FUNCTION_BLOCK "Gr050_Code"	// FB 150
TITLE = Gr050 Machine FB44, FB47, FB50, FB51, FB52, FB56, FB88
//COPYRIGHT:    (C) 1999  BUHLER AG, CH-9240 UZWIL, SWITZERLAND
//
//PRODUCT:      DEFAULT
//
//TITLE:        Machine FB44, FB47, FB50, FB51, FB52, FB56, FB88
//                Machine group control
//                Maschinengruppensteuerung
// 
//--------------------------------------------------------------------------------
// 
//IDENT:        AUTHOR:             DEPT:                              DATE:
// 
//P01_FB150.1.0 A_Egli              CT3                                24.Jul.2008
//             1st Release
// 
//--------------------------------------------------------------------------------
// 
//PURPOSE: 
// 
//MANUAL : 
// 
//RESTRICTIONS: 
// 
//--------------------------------------------------------------------------------
//
AUTHOR : EA
FAMILY : USW
VERSION : 9.9
VAR
  Gr : FB 10;	//Standard interface to group
  InOutValue1 : DINT ;	//Data for user
  InOutValue2 : DINT ;	//Data for user
  OutWayConflict : BOOL ;	//Data for user
  OutSelectionOk : BOOL ;	//Data for user
  CmdNewValue : BOOL ;	//Data for user
  CmdNewJob : BOOL ;	//Data for user
  OutCodeOK : BOOL ;	//Data for user
  InEndOfJob : BOOL ;	//Data for user
  staWayOk : BOOL ;	//Data for user
  EdgeStartRelease : BOOL ;	//Data for user
  USW8 : BOOL ;	//Data for user
  USW9 : BOOL ;	//Data for user
  USW10 : BOOL ;	//Data for user
  USW11 : BOOL ;	//Data for user
  USW12 : BOOL ;	//Data for user
  USW13 : BOOL ;	//Data for user
  USW14 : BOOL ;	//Data for user
  USW15 : BOOL ;	//Data for user
  MaFB44 : FB 735;	// Scourer
  MaFB47 : FB 736;	// Pellet
  MaFB48_ALL : FB 709;	// M3HL2
  MaFB48_Carter : FB 710;	// M3HL2
  MaFB48_MTC : FB 711;	// M3HL2
  MaFB48_MTRA : FB 712;	// M3HL2
  MaFB50All : FB 713;	// Motor+6DI
  MaFB50BKT : FB 714;	// Motor+6DI
  MaFB50ELEV : FB 715;	// Motor+6DI
  MaFB50SIEVE : FB 716;	// Motor+6DI
  MaFB51 : FB 718;	// Motor+2DI
  MaFB52 : FB 719;	// Motor+VLS
  MaFB56 : FB 720;	// DischargerA
  _FB56LL : FB 84;	// SubType FB14: DigInpCont
  MaFB50EBM : FB 724;	// Motor+6DI
  MaFB88 : FB 740;	// DischargerFlat
  MaFB88_Door : FB 14;	// DigInpCont
END_VAR
VAR_TEMP
  tmpEnable : BOOL ;
  tmpFlag : BOOL ;
  tmpCmdNext : BOOL ;
  tmpLocal : BOOL ;
  tmpAspOk : BOOL ;
  tmpHWStop : BOOL ;
  tmpInstanzDBNo : INT ;
END_VAR
BEGIN
NETWORK
TITLE =
NETWORK
TITLE = Read command from group control
NETWORK
TITLE = Call Methode Control
// 1. Handle Interface PCControl      
// 2. Prepare mode --> ModePassive,ModeActive,ModeIdling      
// 3. Reset global flags of the group
      CALL  #Gr (
           FcCode                   := 1);
NETWORK
TITLE = Restart Idling Time
      L     #Gr.Par.ParIdling;
      L     2;
      >=I;
      JC    IdTm;
      T     #Gr.Par.ParIdling;
IdTm: NOP   0;
      CLR;
      S     #Gr.CmdRestartIdling;
NETWORK
TITLE = Prepare global flags
NETWORK
TITLE = Set Pattern (Target position)
NETWORK
TITLE = Interlocking WayOk
NETWORK
TITLE = Interlocking Autostart
      CLR;
      R     #Gr.OutAutostart;
NETWORK
TITLE = Interlocking Enable
      A     #Gr.InEnableGr;
      =     #Gr.OutEnableEl;
NETWORK
TITLE = Interlocking Next
      A     #Gr.CmdNext;
      A     #Gr.OutAutostart;
      AN    #Gr.OutNewWay;
      =     #tmpCmdNext;
NETWORK
TITLE = Interlocking Local / HWStop
      A     "PLC_SystemDB".HardwareStop.General;
      =     #tmpHWStop;
      A     #Gr.ModePassive;
      =     #tmpLocal;
NETWORK
TITLE = MaFB44 : Scourer
      NOP   0;
//-InLocal---
      A     #tmpLocal;
      =     DIX [AR2,P#63.4];
//-Interlocking---
      A     #Gr.OutEnableEl;
      =     DIX [AR2,P#62.0];
// 
      A     #tmpCmdNext;
      S     DIX [AR2,P#63.2];
// 
      A     #Gr.OutSeqStop;
      =     DIX [AR2,P#63.7];
// 
//=Values and commands of elements===
//-FB44Level---
//      CLR
//      S     #MaFB44._FB44Level.CmdRunTimeOutTime
// 
//-Read inputs of elements---
      A     I 2.3;
      =     DIX [AR2,P#72.6];
      A     #tmpHWStop;
      =     DIX [AR2,P#74.0];
      A     I 1.3;
      =     DIX [AR2,P#106.6];
      A     #tmpHWStop;
      =     DIX [AR2,P#108.0];
      A     I 1.5;
      =     DIX [AR2,P#140.6];
      A     #tmpHWStop;
      =     DIX [AR2,P#142.0];
      A     I 2.2;
      =     DIX [AR2,P#174.5];
      A     I 2.1;
      =     DIX [AR2,P#174.6];
      A     #tmpHWStop;
      =     DIX [AR2,P#176.0];
      A     I 2.4;
      =     DIX [AR2,P#208.6];
      A     #tmpHWStop;
      =     DIX [AR2,P#210.0];
      A     I 0.4;
      =     DIX [AR2,P#242.6];
      A     #tmpHWStop;
      =     DIX [AR2,P#244.0];
      A     #tmpHWStop;
      =     DIX [AR2,P#278.0];
// 
//-Set Parameters---
// 
//-Call object control---
      BLD   14;
// 
//-Write outputs---
      =     L 10.0;
      L     DINO;
      T     LW 8;
      CDB;
      OPN   DI [LW 8];
      TAR2  LD 4;
      +AR2  P#60.0;
      UC    FB 735;
      LAR2  LD 4;
      CDB;
      BLD   15;
      A     DIX [AR2,P#74.6];
      =     Q 2.4;
      A     DIX [AR2,P#108.6];
      =     Q 1.1;
      A     DIX [AR2,P#142.6];
      =     Q 2.5;
      A     DIX [AR2,P#176.6];
      =     Q 4.1;
      A     DIX [AR2,P#244.6];
      =     Q 0.7;
      A     DIX [AR2,P#278.7];
      =     Q 4.4;
NETWORK
TITLE = MaFB47 : Pellet Cooler
      NOP   0;
//-InLocal---
      A     #tmpLocal;
      =     DIX [AR2,P#311.4];
// 
//-Interlocking---
      A(;
      O     DIX [AR2,P#65.2];
      O     DIX [AR2,P#65.6];
      );
      A     #Gr.OutEnableEl;
      AN    #Gr.OutSeqStop;
      =     DIX [AR2,P#310.0];
// 
      A     #tmpCmdNext;
      S     DIX [AR2,P#311.2];
// 
//-Additional commands---
      CLR;
      =     DIX [AR2,P#310.1];
      =     DIX [AR2,P#310.2];
      =     DIX [AR2,P#310.3];
      =     DIX [AR2,P#310.4];
      S     DIX [AR2,P#310.5];
// 
//=Values and commands of elements===
// 
//-Values and parameters---
      L     0;
      T     DIW [AR2,P#332.0];
//-FB47Level---
//      CLR
//      S     #MaFB47._FB47Level.CmdRunTimeOutTime
// 
//-Read inputs of elements---
      A     #tmpHWStop;
      =     DIX [AR2,P#328.0];
      A     DIX [AR2,P#388.6];
      =     DIX [AR2,P#386.6];
      A     #tmpHWStop;
      =     DIX [AR2,P#388.0];
      A     I 13.3;
      =     DIX [AR2,P#420.6];
      A     #tmpHWStop;
      =     DIX [AR2,P#422.0];
// 
//-Set Parameters---
// 
//-Call object control---
      BLD   14;
// 
//-Write outputs---
      =     L 10.0;
      L     DINO;
      T     LW 8;
      CDB;
      OPN   DI [LW 8];
      TAR2  LD 4;
      +AR2  P#308.0;
      UC    FB 736;
      LAR2  LD 4;
      CDB;
      BLD   15;
      A     DIX [AR2,P#328.7];
      =     #tmpFlag;
NETWORK
TITLE = MaFB48_ALL : 3 Motors and 2 HL
      NOP   0;
//-InLocal---
      A     #tmpLocal;
      =     DIX [AR2,P#455.4];
// 
//-Interlocking---
      A(;
      O     DIX [AR2,P#313.2];
      O     DIX [AR2,P#313.5];
      O     DIX [AR2,P#313.6];
      );
      A     #Gr.OutEnableEl;
      =     DIX [AR2,P#454.0];
// 
      A     #tmpCmdNext;
      S     DIX [AR2,P#455.2];
// 
      A     #Gr.OutSeqStop;
      =     DIX [AR2,P#455.7];
// 
//-Additional commands---
      CLR;
      =     DIX [AR2,P#454.1];
      CLR;
      =     DIX [AR2,P#454.2];
// 
//=Values and commands of elements===
//-FB48HLLow---
//      CLR
//      S     #MaFB48_ALL._FB48HLLow.CmdRunTimeOutTime
//-FB48HLInlet---
//      CLR
//      S     #MaFB48_ALL._FB48HLInlet.CmdRunTimeOutTime
// 
//-Read inputs of elements---
      A     DIX [AR2,P#466.6];
      =     DIX [AR2,P#464.6];
      A     #tmpHWStop;
      =     DIX [AR2,P#466.0];
      A     DIX [AR2,P#500.6];
      =     DIX [AR2,P#498.6];
      A     #tmpHWStop;
      =     DIX [AR2,P#500.0];
      A     DIX [AR2,P#534.6];
      =     DIX [AR2,P#532.6];
      A     #tmpHWStop;
      =     DIX [AR2,P#534.0];
      AN    I 6.7;
      =     DIX [AR2,P#566.6];
      A     #tmpHWStop;
      =     DIX [AR2,P#568.0];
      AN    I 7.5;
      =     DIX [AR2,P#600.6];
      A     #tmpHWStop;
      =     DIX [AR2,P#602.0];
      A     #tmpHWStop;
      =     DIX [AR2,P#636.0];
// 
//-Set Parameters---
// 
//-Call object control---
      BLD   14;
// 
//-Write outputs---
      =     L 10.0;
      L     DINO;
      T     LW 8;
      CDB;
      OPN   DI [LW 8];
      TAR2  LD 4;
      +AR2  P#452.0;
      UC    FB 709;
      LAR2  LD 4;
      CDB;
      BLD   15;
      A     DIX [AR2,P#636.7];
      =     Q 0.1;
NETWORK
TITLE = MaFB48_Carter : 3 Motors and 2 HL
      NOP   0;
//-InLocal---
      A     #tmpLocal;
      =     DIX [AR2,P#669.4];
// 
//-Interlocking---
      A     DIX [AR2,P#457.2];
      A     #Gr.OutEnableEl;
      =     DIX [AR2,P#668.0];
// 
      A     #tmpCmdNext;
      S     DIX [AR2,P#669.2];
// 
      A     #Gr.OutSeqStop;
      =     DIX [AR2,P#669.7];
// 
//-Additional commands---
      CLR;
      =     DIX [AR2,P#668.1];
      CLR;
      =     DIX [AR2,P#668.2];
// 
//=Values and commands of elements===
//-FB48HLLow_C---
//      CLR
//      S     #MaFB48_Carter._FB48HLLow_C.CmdRunTimeOutTime
//-FB48HLInlet_C---
//      CLR
//      S     #MaFB48_Carter._FB48HLInlet_C.CmdRunTimeOutTime
// 
//-Read inputs of elements---
      A     I 10.0;
      =     DIX [AR2,P#678.6];
      A     #tmpHWStop;
      =     DIX [AR2,P#680.0];
      A     I 9.7;
      =     DIX [AR2,P#712.6];
      A     #tmpHWStop;
      =     DIX [AR2,P#714.0];
      A     I 12.3;
      =     DIX [AR2,P#746.6];
      A     #tmpHWStop;
      =     DIX [AR2,P#748.0];
      AN    I 6.6;
      =     DIX [AR2,P#780.6];
      A     #tmpHWStop;
      =     DIX [AR2,P#782.0];
      AN    I 8.0;
      =     DIX [AR2,P#814.6];
      A     #tmpHWStop;
      =     DIX [AR2,P#816.0];
      A     #tmpHWStop;
      =     DIX [AR2,P#850.0];
// 
//-Set Parameters---
// 
//-Call object control---
      BLD   14;
// 
//-Write outputs---
      =     L 10.0;
      L     DINO;
      T     LW 8;
      CDB;
      OPN   DI [LW 8];
      TAR2  LD 4;
      +AR2  P#666.0;
      UC    FB 710;
      LAR2  LD 4;
      CDB;
      BLD   15;
      A     DIX [AR2,P#680.6];
      =     Q 4.3;
      A     DIX [AR2,P#714.6];
      =     Q 4.6;
      A     DIX [AR2,P#748.6];
      =     Q 5.1;
      A     DIX [AR2,P#850.7];
      =     Q 0.1;
NETWORK
TITLE = MaFB48_MTC : 3 Motors and 2 HL
      NOP   0;
//-InLocal---
      A     #tmpLocal;
      =     DIX [AR2,P#883.4];
// 
//-Interlocking---
      A     DIX [AR2,P#671.2];
      A     #Gr.OutEnableEl;
      =     DIX [AR2,P#882.0];
// 
      A     #tmpCmdNext;
      S     DIX [AR2,P#883.2];
// 
      A     #Gr.OutSeqStop;
      =     DIX [AR2,P#883.7];
// 
//-Additional commands---
      CLR;
      =     DIX [AR2,P#882.1];
      CLR;
      =     DIX [AR2,P#882.2];
// 
//=Values and commands of elements===
//-FB48HLLow---
//      CLR
//      S     #MaFB48_MTC._FB48HLLow.CmdRunTimeOutTime
//-FB48HLInletMTC---
//      CLR
//      S     #MaFB48_MTC._FB48HLInletMTC.CmdRunTimeOutTime
// 
//-Read inputs of elements---
      A     I 7.7;
      =     DIX [AR2,P#892.6];
      A     #tmpHWStop;
      =     DIX [AR2,P#894.0];
      A     I 12.7;
      =     DIX [AR2,P#926.6];
      A     #tmpHWStop;
      =     DIX [AR2,P#928.0];
      A     I 8.1;
      =     DIX [AR2,P#960.6];
      A     #tmpHWStop;
      =     DIX [AR2,P#962.0];
      AN    I 6.7;
      =     DIX [AR2,P#994.6];
      A     #tmpHWStop;
      =     DIX [AR2,P#996.0];
      AN    I 7.6;
      =     DIX [AR2,P#1028.6];
      A     #tmpHWStop;
      =     DIX [AR2,P#1030.0];
      A     #tmpHWStop;
      =     DIX [AR2,P#1064.0];
// 
//-Set Parameters---
// 
//-Call object control---
      BLD   14;
// 
//-Write outputs---
      =     L 10.0;
      L     DINO;
      T     LW 8;
      CDB;
      OPN   DI [LW 8];
      TAR2  LD 4;
      +AR2  P#880.0;
      UC    FB 711;
      LAR2  LD 4;
      CDB;
      BLD   15;
      A     DIX [AR2,P#894.6];
      =     Q 4.2;
      A     DIX [AR2,P#928.6];
      =     Q 5.2;
      A     DIX [AR2,P#962.6];
      =     Q 3.0;
      A     DIX [AR2,P#1064.7];
      =     Q 0.1;
NETWORK
TITLE = MaFB48_MTRA : 3 Motors and 2 HL
      NOP   0;
//-InLocal---
      A     #tmpLocal;
      =     DIX [AR2,P#1097.4];
// 
//-Interlocking---
      A     DIX [AR2,P#885.2];
      A     #Gr.OutEnableEl;
      =     DIX [AR2,P#1096.0];
// 
      A     #tmpCmdNext;
      S     DIX [AR2,P#1097.2];
// 
      A     #Gr.OutSeqStop;
      =     DIX [AR2,P#1097.7];
// 
//-Additional commands---
      CLR;
      =     DIX [AR2,P#1096.1];
      CLR;
      =     DIX [AR2,P#1096.2];
// 
//=Values and commands of elements===
//-FB48HLInletMTRA---
//      CLR
//      S     #MaFB48_MTRA._FB48HLInletMTRA.CmdRunTimeOutTime
// 
//-Read inputs of elements---
      A     I 12.5;
      =     DIX [AR2,P#1106.6];
      A     #tmpHWStop;
      =     DIX [AR2,P#1108.0];
      A     I 8.3;
      =     DIX [AR2,P#1140.6];
      A     #tmpHWStop;
      =     DIX [AR2,P#1142.0];
      A     DIX [AR2,P#1176.6];
      =     DIX [AR2,P#1174.6];
      A     #tmpHWStop;
      =     DIX [AR2,P#1176.0];
      AN    I 7.4;
      =     DIX [AR2,P#1242.6];
      A     #tmpHWStop;
      =     DIX [AR2,P#1244.0];
// 
//-Set Parameters---
// 
//-Call object control---
      BLD   14;
// 
//-Write outputs---
      =     L 10.0;
      L     DINO;
      T     LW 8;
      CDB;
      OPN   DI [LW 8];
      TAR2  LD 4;
      +AR2  P#1094.0;
      UC    FB 712;
      LAR2  LD 4;
      CDB;
      BLD   15;
      A     DIX [AR2,P#1108.6];
      =     Q 5.0;
      A     DIX [AR2,P#1142.6];
      =     Q 3.1;
NETWORK
TITLE = MaFB50All : Motor + 4 digiatl inputs     
      NOP   0;
//-InLocal---
      A     #tmpLocal;
      =     DIX [AR2,P#1311.4];
//-Interlocking---
      A     DIX [AR2,P#1099.2];
      A     #Gr.OutEnableEl;
      =     DIX [AR2,P#1310.1];
      A     #tmpCmdNext;
      S     DIX [AR2,P#1311.2];
      A     #Gr.OutSeqStop;
      =     DIX [AR2,P#1311.7];
// 
//=Values and commands of elements===
//-FB50Mon1---
//      CLR
//      S     #MaFB50All._FB50Mon1.CmdRunTimeOutTime
//-FB50Mon2---
//      CLR
//      S     #MaFB50All._FB50Mon2.CmdRunTimeOutTime
//-FB50Mon3---
//      CLR
//      S     #MaFB50All._FB50Mon3.CmdRunTimeOutTime
//-FB50MonInlet---
//      CLR
//      S     #MaFB50All._FB50MonInlet.CmdRunTimeOutTime
// 
//-Read inputs of elements---
      A     I 22.0;
      =     DIX [AR2,P#1322.6];
      A     #tmpHWStop;
      =     DIX [AR2,P#1324.0];
      A     I 22.1;
      =     DIX [AR2,P#1356.6];
      A     #tmpHWStop;
      =     DIX [AR2,P#1358.0];
      A     I 22.2;
      =     DIX [AR2,P#1390.6];
      A     #tmpHWStop;
      =     DIX [AR2,P#1392.0];
      A     I 22.3;
      =     DIX [AR2,P#1424.6];
      A     #tmpHWStop;
      =     DIX [AR2,P#1426.0];
      A     I 22.4;
      =     DIX [AR2,P#1526.6];
      A     I 22.5;
      =     DIX [AR2,P#1526.5];
      A     #tmpHWStop;
      =     DIX [AR2,P#1528.0];
// 
//-Set Parameters---
// 
//-Call object control---
      BLD   14;
// 
//-Write outputs---
      =     L 10.0;
      L     DINO;
      T     LW 8;
      CDB;
      OPN   DI [LW 8];
      TAR2  LD 4;
      +AR2  P#1308.0;
      UC    FB 713;
      LAR2  LD 4;
      CDB;
      BLD   15;
      A     DIX [AR2,P#1528.6];
      =     Q 22.4;
      A     DIX [AR2,P#1528.5];
      =     Q 22.5;
NETWORK
TITLE = MaFB50BKT : Motor + 4 digiatl inputs
      NOP   0;
//-InLocal---
      A     #tmpLocal;
      =     DIX [AR2,P#1561.4];
//-Interlocking---
      A     DIX [AR2,P#1313.2];
      A     #Gr.OutEnableEl;
      =     DIX [AR2,P#1560.1];
      A     #tmpCmdNext;
      S     DIX [AR2,P#1561.2];
      A     #Gr.OutSeqStop;
      =     DIX [AR2,P#1561.7];
// 
//=Values and commands of elements===
//-FB50LSBKT---
//      CLR
//      S     #MaFB50BKT._FB50LSBKT.CmdRunTimeOutTime
//-FB50SM1BKT---
//      CLR
//      S     #MaFB50BKT._FB50SM1BKT.CmdRunTimeOutTime
//-FB50SM2BKT---
//      CLR
//      S     #MaFB50BKT._FB50SM2BKT.CmdRunTimeOutTime
//-FB50HLBKT---
//      CLR
//      S     #MaFB50BKT._FB50HLBKT.CmdRunTimeOutTime
// 
//-Read inputs of elements---
      A     I 13.5;
      =     DIX [AR2,P#1572.6];
      A     #tmpHWStop;
      =     DIX [AR2,P#1574.0];
      A     I 1.4;
      =     DIX [AR2,P#1606.6];
      A     #tmpHWStop;
      =     DIX [AR2,P#1608.0];
      A     I 1.2;
      =     DIX [AR2,P#1640.6];
      A     #tmpHWStop;
      =     DIX [AR2,P#1642.0];
      A     I 8.2;
      =     DIX [AR2,P#1674.6];
      A     #tmpHWStop;
      =     DIX [AR2,P#1676.0];
      A     I 12.4;
      =     DIX [AR2,P#1776.6];
      A     I 12.2;
      =     DIX [AR2,P#1776.5];
      A     #tmpHWStop;
      =     DIX [AR2,P#1778.0];
// 
//-Set Parameters---
// 
//-Call object control---
      BLD   14;
// 
//-Write outputs---
      =     L 10.0;
      L     DINO;
      T     LW 8;
      CDB;
      OPN   DI [LW 8];
      TAR2  LD 4;
      +AR2  P#1558.0;
      UC    FB 714;
      LAR2  LD 4;
      CDB;
      BLD   15;
      A     DIX [AR2,P#1778.6];
      =     Q 3.4;
      A     DIX [AR2,P#1778.5];
      =     Q 3.5;
NETWORK
TITLE = MaFB50SIEVE : Motor + 4 digiatl inputs
      NOP   0;
//-InLocal---
      A     #tmpLocal;
      =     DIX [AR2,P#2061.4];
//-Interlocking---
      A     DIX [AR2,P#1563.2];
      A     #Gr.OutEnableEl;
      =     DIX [AR2,P#2060.1];
      A     #tmpCmdNext;
      S     DIX [AR2,P#2061.2];
      A     #Gr.OutSeqStop;
      =     DIX [AR2,P#2061.7];
// 
//=Values and commands of elements===
//-FB50HL_Waste---
//      CLR
//      S     #MaFB50SIEVE._FB50HL_Waste.CmdRunTimeOutTime
//-FB50LSA---
//      CLR
//      S     #MaFB50SIEVE._FB50LSA.CmdRunTimeOutTime
//-FB50LSB---
//      CLR
//      S     #MaFB50SIEVE._FB50LSB.CmdRunTimeOutTime
//-FB50HL_Sieve---
//      CLR
//      S     #MaFB50SIEVE._FB50HL_Sieve.CmdRunTimeOutTime
// 
//-Read inputs of elements---
      A     I 28.5;
      =     DIX [AR2,P#2072.6];
      A     #tmpHWStop;
      =     DIX [AR2,P#2074.0];
      A     I 9.5;
      =     DIX [AR2,P#2106.6];
      A     #tmpHWStop;
      =     DIX [AR2,P#2108.0];
      A     I 0.0;
      =     DIX [AR2,P#2140.6];
      A     #tmpHWStop;
      =     DIX [AR2,P#2142.0];
      A     I 8.6;
      =     DIX [AR2,P#2174.6];
      A     #tmpHWStop;
      =     DIX [AR2,P#2176.0];
      A     I 10.3;
      =     DIX [AR2,P#2276.6];
      A     I 10.1;
      =     DIX [AR2,P#2276.5];
      A     #tmpHWStop;
      =     DIX [AR2,P#2278.0];
// 
//-Set Parameters---
// 
//-Call object control---
      BLD   14;
// 
//-Write outputs---
      =     L 10.0;
      L     DINO;
      T     LW 8;
      CDB;
      OPN   DI [LW 8];
      TAR2  LD 4;
      +AR2  P#2058.0;
      UC    FB 716;
      LAR2  LD 4;
      CDB;
      BLD   15;
      A     DIX [AR2,P#2278.6];
      =     Q 3.6;
      A     DIX [AR2,P#2278.5];
      =     Q 3.3;
NETWORK
TITLE = MaFB51 : Motor with 2 digital input
      NOP   0;
//-InLocal---
      A     #tmpLocal;
      =     DIX [AR2,P#2311.4];
// 
//-Interlocking---
      A     #Gr.OutEnableEl;
      =     DIX [AR2,P#2310.1];
// 
      A     DIX [AR2,P#2063.2];
      A     #tmpCmdNext;
      S     DIX [AR2,P#2311.2];
// 
      A     #Gr.OutSeqStop;
      =     DIX [AR2,P#2311.7];
// 
//=Values and commands of elements===
//-FB51Mon1---
//      CLR
//      S     #MaFB51._FB51Mon1.CmdRunTimeOutTime
//-FB51Mon2---
//      CLR
//      S     #MaFB51._FB51Mon2.CmdRunTimeOutTime
// 
//-Read inputs of elements---
      AN    I 0.3;
      =     DIX [AR2,P#2320.6];
      A     #tmpHWStop;
      =     DIX [AR2,P#2322.0];
      AN    I 0.5;
      =     DIX [AR2,P#2354.6];
      A     #tmpHWStop;
      =     DIX [AR2,P#2356.0];
// 
//-Set Parameters---
// 
//-Call object control---
      BLD   14;
// 
//-Write outputs---
      =     L 10.0;
      L     DINO;
      T     LW 8;
      CDB;
      OPN   DI [LW 8];
      TAR2  LD 4;
      +AR2  P#2308.0;
      UC    FB 718;
      LAR2  LD 4;
      CDB;
      BLD   15;
NETWORK
TITLE = MaFB52 : Motor with Bypass flap
      NOP   0;
//-InLocal---
      A     #tmpLocal;
      =     DIX [AR2,P#2423.4];
//-Interlocking---
      A     #Gr.OutEnableEl;
      =     DIX [AR2,P#2422.1];
      A     #tmpCmdNext;
      S     DIX [AR2,P#2423.2];
      A     #Gr.OutSeqStop;
      =     DIX [AR2,P#2423.7];
      A     "ENG_RemarkFlag";
      =     DIX [AR2,P#2422.4];
//-Additional commands---
      CLR;
      =     DIX [AR2,P#2422.2];
      =     DIX [AR2,P#2422.3];
// 
//=Values and commands of elements===
//-FB52Mon1---
//      CLR
//      S     #MaFB52._FB52Mon1.CmdRunTimeOutTime
//-FB52HLInlet---
//      CLR
//      S     #MaFB52._FB52HLInlet.CmdRunTimeOutTime
// 
//-Read inputs of elements---
      A     I 52.1;
      =     DIX [AR2,P#2438.6];
      A     #tmpHWStop;
      =     DIX [AR2,P#2440.0];
      A     I 33.4;
      =     DIX [AR2,P#2472.6];
      A     I 33.3;
      =     DIX [AR2,P#2472.5];
      A     #tmpHWStop;
      =     DIX [AR2,P#2474.0];
      A     I 52.3;
      =     DIX [AR2,P#2506.5];
      A     I 52.4;
      =     DIX [AR2,P#2506.6];
      A     #tmpHWStop;
      =     DIX [AR2,P#2508.0];
      AN    I 52.0;
      =     DIX [AR2,P#2540.6];
      A     #tmpHWStop;
      =     DIX [AR2,P#2542.0];
      A     I 52.6;
      =     DIX [AR2,P#2574.5];
      A     I 52.7;
      =     DIX [AR2,P#2574.6];
      A     #tmpHWStop;
      =     DIX [AR2,P#2576.0];
      A     #tmpHWStop;
      =     DIX [AR2,P#2610.0];
// 
//-Set Parameters---
// 
//-Call object control---
      BLD   14;
// 
//-Write outputs---
      =     L 10.0;
      L     DINO;
      T     LW 8;
      CDB;
      OPN   DI [LW 8];
      TAR2  LD 4;
      +AR2  P#2420.0;
      UC    FB 719;
      LAR2  LD 4;
      CDB;
      BLD   15;
      A     DIX [AR2,P#2474.6];
      =     Q 36.4;
      A     DIX [AR2,P#2474.5];
      =     Q 36.3;
      A     DIX [AR2,P#2508.5];
      =     Q 52.3;
      A     DIX [AR2,P#2508.6];
      =     Q 52.4;
      A     DIX [AR2,P#2576.5];
      =     Q 52.6;
      A     DIX [AR2,P#2576.6];
      =     Q 52.7;
NETWORK
TITLE = MaFB56 : Bin Discharger A
      NOP   0;
//-InLocal---
      A     #tmpLocal;
      =     DIX [AR2,P#2643.4];
// 
//-Interlocking---
      A     #Gr.OutEnableEl;
      AN    #Gr.OutSeqStop;
      =     DIX [AR2,P#2642.0];
// 
      A     #tmpCmdNext;
      S     DIX [AR2,P#2643.2];
// 
//=Additional commands and signals===
//-Bin emptying---
      CLR;
      =     DIX [AR2,P#2642.1];
//-Low Level---
      A     DIX [AR2,P#2769.0];
      O     DIX [AR2,P#2769.1];
      O     DIX [AR2,P#2769.4];
      =     DIX [AR2,P#2642.3];
      A     DIX [AR2,P#2769.2];
      =     DIX [AR2,P#2642.4];
// 
//=Values and commands of elements===
//-FB56LS---
//      CLR
//      S     #MaFB56._FB56LS.CmdRunTimeOutTime
// 
//-Read inputs of elements---
      A     I 33.6;
      =     DIX [AR2,P#2664.6];
      A     I 34.1;
      =     DIX [AR2,P#2664.5];
      A     I 34.0;
      =     DIX [AR2,P#2664.3];
      A     I 33.7;
      =     DIX [AR2,P#2664.4];
      A     #tmpHWStop;
      =     DIX [AR2,P#2666.0];
      A     I 34.2;
      =     DIX [AR2,P#2698.6];
      A     #tmpHWStop;
      =     DIX [AR2,P#2700.0];
      A     #tmpHWStop;
      =     DIX [AR2,P#2734.0];
// 
//-Set Parameters---
// 
//-Call object control---
      BLD   14;
// 
//-Write outputs---
      =     L 10.0;
      L     DINO;
      T     LW 8;
      CDB;
      OPN   DI [LW 8];
      TAR2  LD 4;
      +AR2  P#2640.0;
      UC    FB 720;
      LAR2  LD 4;
      CDB;
      BLD   15;
      A     DIX [AR2,P#2666.6];
      =     Q 36.1;
      A     DIX [AR2,P#2666.5];
      =     Q 35.0;
      A     DIX [AR2,P#2666.3];
      =     Q 36.0;
      A     DIX [AR2,P#2666.4];
      =     Q 36.2;
      A     DIX [AR2,P#2700.6];
      =     Q 35.3;
NETWORK
TITLE = FB56LL : 
      NOP   0;
//-Local---
      SET;
      =     DIX [AR2,P#2767.4];
// 
//-Monitoring---
// 
//-Read inputs---
      A     #tmpHWStop;
      =     DIX [AR2,P#2768.0];
// 
//-Set Parameters---
// 
//-Call object control---
      BLD   14;
// 
//-Write outputs---
      =     L 10.0;
      L     DINO;
      T     LW 8;
      CDB;
      OPN   DI [LW 8];
      TAR2  LD 4;
      +AR2  P#2764.0;
      UC    "GCS7_E_Level";
      LAR2  LD 4;
      CDB;
      BLD   15;
NETWORK
TITLE = MaFB50ELEV : Motor + 4 digiatl inputs 
      NOP   0;
//-InLocal---
      A     #tmpLocal;
      =     DIX [AR2,P#1811.4];
//-Interlocking---
      A     DIX [AR2,P#2645.2];
      A     #Gr.OutEnableEl;
      =     DIX [AR2,P#1810.1];
      A     #tmpCmdNext;
      S     DIX [AR2,P#1811.2];
      A     #Gr.OutSeqStop;
      =     DIX [AR2,P#1811.7];
// 
//=Values and commands of elements===
//-FB50BM1---
//      CLR
//      S     #MaFB50ELEV._FB50BM1.CmdRunTimeOutTime
//-FB50BM2---
//      CLR
//      S     #MaFB50ELEV._FB50BM2.CmdRunTimeOutTime
//-FB50SM_ELEV---
//      CLR
//      S     #MaFB50ELEV._FB50SM_ELEV.CmdRunTimeOutTime
// 
//-Read inputs of elements---
      A     I 9.0;
      =     DIX [AR2,P#1856.6];
      A     #tmpHWStop;
      =     DIX [AR2,P#1858.0];
      A     I 8.7;
      =     DIX [AR2,P#1890.6];
      A     #tmpHWStop;
      =     DIX [AR2,P#1892.0];
      A     I 2.5;
      =     DIX [AR2,P#1924.6];
      A     #tmpHWStop;
      =     DIX [AR2,P#1926.0];
      A     I 12.6;
      =     DIX [AR2,P#2026.6];
      A     I 13.4;
      =     DIX [AR2,P#2026.5];
      A     #tmpHWStop;
      =     DIX [AR2,P#2028.0];
// 
//-Set Parameters---
// 
//-Call object control---
      BLD   14;
// 
//-Write outputs---
      =     L 10.0;
      L     DINO;
      T     LW 8;
      CDB;
      OPN   DI [LW 8];
      TAR2  LD 4;
      +AR2  P#1808.0;
      UC    FB 715;
      LAR2  LD 4;
      CDB;
      BLD   15;
      A     DIX [AR2,P#2028.6];
      =     Q 13.7;
      A     DIX [AR2,P#2028.5];
      =     Q 14.4;
NETWORK
TITLE = MaFB50EBM : Elevator mit EBM
      NOP   0;
//-Read Inputs of Machine---
      A     I 150.0;
      =     DIX [AR2,P#2800.6];
//-InLocal---
      A     #tmpLocal;
      =     DIX [AR2,P#2801.4];
//-Interlocking---
      A     DIX [AR2,P#1813.2];
      A     #Gr.OutEnableEl;
      =     DIX [AR2,P#2800.1];
      A     #tmpCmdNext;
      S     DIX [AR2,P#2801.2];
      A     #Gr.OutSeqStop;
      =     DIX [AR2,P#2801.7];
// 
//-Additional commands---
      A     DIX [AR2,P#2848.6];
      O     DIX [AR2,P#2882.6];
      O     DIX [AR2,P#2916.6];
      O     DIX [AR2,P#2950.6];
      O     DIX [AR2,P#2984.6];
      A(;
      O     DIX [AR2,P#3017.5];
      O     DIX [AR2,P#2801.4];
      );
      A     DIX [AR2,P#2803.4];
      S     DIX [AR2,P#2801.3];
// 
//=Values and commands of elements===
//-MaFB50BMTop1---
//      CLR
//      S     #MaFB50EBM.MaFB50BMTop1.CmdRunTimeOutTime
//-MaFB50BMTop2---
//      CLR
//      S     #MaFB50EBM.MaFB50BMTop2.CmdRunTimeOutTime
//-MaFB50BMBottom1---
//      CLR
//      S     #MaFB50EBM.MaFB50BMBottom1.CmdRunTimeOutTime
//-MaFB50BMBottom2---
//      CLR
//      S     #MaFB50EBM.MaFB50BMBottom2.CmdRunTimeOutTime
//-MaFB50SM---
//      CLR
//      S     #MaFB50EBM.MaFB50SM.CmdRunTimeOutTime
// 
//-Read inputs of elements---
      A     I 150.1;
      =     DIX [AR2,P#2846.6];
      A     #tmpHWStop;
      =     DIX [AR2,P#2848.0];
      A     I 150.2;
      =     DIX [AR2,P#2880.6];
      A     #tmpHWStop;
      =     DIX [AR2,P#2882.0];
      A     I 150.4;
      =     DIX [AR2,P#2914.6];
      A     #tmpHWStop;
      =     DIX [AR2,P#2916.0];
      A     I 150.5;
      =     DIX [AR2,P#2948.6];
      A     #tmpHWStop;
      =     DIX [AR2,P#2950.0];
      A     I 150.3;
      =     DIX [AR2,P#2982.6];
      A     #tmpHWStop;
      =     DIX [AR2,P#2984.0];
      A     I 149.0;
      =     DIX [AR2,P#3016.6];
      A     #tmpHWStop;
      =     DIX [AR2,P#3018.0];
// 
//-Set Parameters---
// 
//-Call object control---
      BLD   14;
// 
//-Write outputs---
      =     L 10.0;
      L     DINO;
      T     LW 8;
      CDB;
      OPN   DI [LW 8];
      TAR2  LD 4;
      +AR2  P#2798.0;
      UC    FB 724;
// 
      LAR2  LD 4;
      CDB;
      BLD   15;
      A     DIX [AR2,P#2802.7];
      =     Q 150.0;
      A     DIX [AR2,P#2802.4];
      =     Q 150.1;
      A     DIX [AR2,P#2802.5];
// 
      =     Q 150.2;
      A     DIX [AR2,P#2802.6];
      =     Q 150.3;
      AN    DIX [AR2,P#2849.4];
      AN    DIX [AR2,P#2883.4];
      AN    DIX [AR2,P#2917.4];
      AN    DIX [AR2,P#2951.4];
      AN    DIX [AR2,P#2985.4];
      ON    DIX [AR2,P#2801.4];
      O     DIX [AR2,P#3017.5];
      =     Q 150.4;
      A     DIX [AR2,P#3018.6];
      =     Q 149.0;
NETWORK
TITLE = MaFB88_Door : Bin Discharger Flat-Bottom
      NOP   0;
//-InLocal---
      A     #tmpLocal;
      =     DIX [AR2,P#3343.4];
// 
//-Monitoring---
      SET;
      =     DIX [AR2,P#3342.0];
      CLR;
      =     DIX [AR2,P#3342.1];
// 
//-PreAlarm---
      CLR;
      =     DIX [AR2,P#3342.2];
      CLR;
      =     DIX [AR2,P#3342.3];
// 
//-Additional commands---
//      CLR
//      S     #MaFB88_Door.CmdRunTimeOutTime
// 
//-Read inputs---
      A     I 96.2;
      =     DIX [AR2,P#3342.6];
      A     #tmpHWStop;
      =     DIX [AR2,P#3344.0];
// 
//-Set Parameters---
// 
//-Call object control---
      BLD   14;
// 
//-Write outputs---
      =     L 10.0;
      L     DINO;
      T     LW 8;
      CDB;
      OPN   DI [LW 8];
      TAR2  LD 4;
      +AR2  P#3340.0;
      UC    "GCS7_E_DigInput";
      LAR2  LD 4;
      CDB;
      BLD   15;
NETWORK
TITLE = MaFB88 : Bin Discharger Flat-Bottom  
      NOP   0;
//-InLocal---
// 
//-Interlocking---
// 
      SET;
      S     DIX [AR2,P#3051.2];
// 
//=Additional commands and signals===
//-Bin emptying---
//-LSDorr---
      A     DIX [AR2,P#3345.0];
      =     DIX [AR2,P#3050.6];
      A     DIX [AR2,P#3345.2];
      =     DIX [AR2,P#3050.5];
// 
//=Values and commands of elements===
//-MaFB88_LL---
//      CLR
//      S     #MaFB88.MaFB88_LL.CmdRunTimeOutTime
//-MaFB88_Switch---
//      CLR
//      S     #MaFB88.MaFB88_Switch.CmdRunTimeOutTime
// 
//-Read inputs of elements---
      A     I 95.0;
      =     DIX [AR2,P#3070.5];
      A     I 95.1;
      =     DIX [AR2,P#3070.6];
      A     #tmpHWStop;
      =     DIX [AR2,P#3072.0];
      A     #tmpHWStop;
      =     DIX [AR2,P#3106.0];
      A     I 96.5;
      =     DIX [AR2,P#3104.6];
      A     I 96.3;
      =     DIX [AR2,P#3138.6];
      A     #tmpHWStop;
      =     DIX [AR2,P#3140.0];
      A     I 96.4;
      =     DIX [AR2,P#3172.6];
      A     #tmpHWStop;
      =     DIX [AR2,P#3174.0];
      A     I 95.2;
      =     DIX [AR2,P#3206.5];
      A     I 95.3;
      =     DIX [AR2,P#3206.6];
      A     #tmpHWStop;
      =     DIX [AR2,P#3208.0];
      A     I 95.4;
      =     DIX [AR2,P#3240.5];
      A     I 95.5;
      =     DIX [AR2,P#3240.6];
      A     #tmpHWStop;
      =     DIX [AR2,P#3242.0];
      A     I 95.6;
      =     DIX [AR2,P#3274.5];
      A     I 95.7;
      =     DIX [AR2,P#3274.6];
      A     #tmpHWStop;
      =     DIX [AR2,P#3276.0];
      A     I 96.0;
      =     DIX [AR2,P#3308.5];
      A     I 96.1;
      =     DIX [AR2,P#3308.6];
      A     #tmpHWStop;
      =     DIX [AR2,P#3310.0];
// 
//-Set Parameters---
// 
//-Call object control---
      BLD   14;
// 
//-Write outputs---
      =     L 10.0;
      L     DINO;
      T     LW 8;
      CDB;
      OPN   DI [LW 8];
      TAR2  LD 4;
      +AR2  P#3048.0;
      UC    FB 740;
      LAR2  LD 4;
      CDB;
      BLD   15;
      A     DIX [AR2,P#3072.6];
      =     Q 95.0;
      A     DIX [AR2,P#3140.6];
      =     Q 96.3;
NETWORK
TITLE = Test Fault
      A     DIX [AR2,P#65.4];
      O     DIX [AR2,P#313.4];
      O     DIX [AR2,P#457.4];
      O     DIX [AR2,P#671.4];
      O     DIX [AR2,P#885.4];
      O     DIX [AR2,P#1099.4];
      O     DIX [AR2,P#1313.4];
      O     DIX [AR2,P#1563.4];
      O     DIX [AR2,P#2063.4];
      O     DIX [AR2,P#2313.4];
      O     DIX [AR2,P#2425.4];
      O     DIX [AR2,P#2645.4];
      O     DIX [AR2,P#2769.4];
      O     DIX [AR2,P#1813.4];
      O     DIX [AR2,P#2803.4];
      O     DIX [AR2,P#3345.4];
      O     DIX [AR2,P#3053.4];
      =     #Gr.VarFault;
NETWORK
TITLE = Test Warning
      A     DIX [AR2,P#2312.0];
      =     #Gr.OutWarning;
NETWORK
TITLE = Test Stopped
      A     DIX [AR2,P#65.0];
      A(;
      O     DIX [AR2,P#313.0];
      O     DIX [AR2,P#313.6];
      );
      A     DIX [AR2,P#457.0];
      A     DIX [AR2,P#671.0];
      A     DIX [AR2,P#885.0];
      A     DIX [AR2,P#1099.0];
      A     DIX [AR2,P#1313.0];
      A     DIX [AR2,P#1563.0];
      A     DIX [AR2,P#2063.0];
      A     DIX [AR2,P#2313.0];
      A(;
      AN    DIX [AR2,P#2422.1];
      O     DIX [AR2,P#2423.7];
      A     DIX [AR2,P#2425.6];
      O     DIX [AR2,P#2425.0];
      );
      A     DIX [AR2,P#2645.0];
      A     DIX [AR2,P#1813.0];
      A     DIX [AR2,P#2803.0];
      A     DIX [AR2,P#3053.0];
      AN    #Gr.VarFault;
      =     #Gr.VarStopped;
NETWORK
TITLE = Test Started
      A(;
      O     DIX [AR2,P#65.6];
      O     DIX [AR2,P#65.2];
      );
      A(;
      O     DIX [AR2,P#313.2];
      O     DIX [AR2,P#313.5];
      O     DIX [AR2,P#313.6];
      );
      A     DIX [AR2,P#457.2];
      A     DIX [AR2,P#671.2];
      A     DIX [AR2,P#885.2];
      A     DIX [AR2,P#1099.2];
      A(;
      O     DIX [AR2,P#1313.2];
      O     DIX [AR2,P#1313.5];
      );
      A(;
      O     DIX [AR2,P#1563.2];
      O     DIX [AR2,P#1563.5];
      );
      A(;
      O     DIX [AR2,P#2063.2];
      O     DIX [AR2,P#2063.5];
      );
      A(;
      O     DIX [AR2,P#2313.2];
      O     DIX [AR2,P#2313.5];
      );
      A(;
      A     DIX [AR2,P#2422.1];
      AN    DIX [AR2,P#2423.7];
      A     DIX [AR2,P#2425.6];
      O     DIX [AR2,P#2425.2];
      O     DIX [AR2,P#2425.5];
      );
      A     DIX [AR2,P#2645.2];
      A(;
      O     DIX [AR2,P#1813.2];
      O     DIX [AR2,P#1813.5];
      );
      A     DIX [AR2,P#2803.2];
      A     DIX [AR2,P#3053.2];
      AN    #Gr.VarStopped;
      AN    #Gr.VarFault;
      =     #Gr.VarStarted;
NETWORK
TITLE = Enable Previous Group
      A     #Gr.VarStarted;
      =     #Gr.OutEnablePrevGr;
NETWORK
TITLE = Call Methode State
//1. Make State of the group: This function use the signals:
//        Gr.VarStopped, Gr.VarStarted, Gr.VarFault
//2.Reset Commands to group: e.g.CmdFaultReset
      CALL  #Gr (
           FcCode                   := 2);
NETWORK
TITLE = Init
      SET;
      R     #CmdNewValue;
      R     #CmdNewJob;
NETWORK
TITLE = Write data to group control
NETWORK
TITLE = End of block
      BE;
END_FUNCTION_BLOCK

FUNCTION_BLOCK "SSA_PneumaticControl_Fct"	// FB 841
TITLE = PNEUMATIC-CONTROLLER
//
//COPYRIGHT:    (C) 2007 BY BUHLER AG
//                          CH-9240 UZWIL  SWITZERLAND
//
//PRODUCT:      GCS7R2_SSA_GP92
//
//TITLE:        Pneumatic controller
//
//              Pneumatic Regler
//
//
// 
//--------------------------------------------------------------------------------
//
//IDENT:         AUTOR:              DEPT:                             DATE:
//SSA_FB841.4.0  Ph. Engler          GP92                              04-Jun-2009
//               - GCS7
//SSA_FB841.3.0  Ph. Engler          GP92                              05-Apr-2009
//               - Changed to a new GCS type
//SSA_FB1811.2.0 Ph. Engler          GP92                              22-Jan-2008
//               - Without StartupTime and StartupSpeed
//SSA_FB1811.1.1 Ph. Engler          GP92                              22-Jan-2008
//               - Immediate change to running in manual mode
//               - Changing to stRunning after startup of the ventilator
//SSA_FB1811.1.0 Ph. Engler          GP92                              04-Dec-2007
//               1st Release
//
//--------------------------------------------------------------------------------
//
//PURPOSE: 
//
//MANUAL : 
//
//RESTRICTIONS:
//
//--------------------------------------------------------------------------------
//
//
//
AUTHOR : PE
FAMILY : SSA
VERSION : 4.0
VAR
  StCode : INT ;
  InEnable : BOOL ;
  InFullLoad : BOOL ;
  CmdFaultReset : BOOL ;
  CmdNewValue : BOOL ;
  CmdNext : BOOL ;	//Pulse to start the element in automatic mode (see global flags)
  spare01 : BOOL ;
  InLocal : BOOL ;
  InManual : BOOL ;
  InNoPressureAlarm : BOOL ;
  InWarning : BOOL ;
  InReport : BOOL ;	//Report of all state transitions
  InHWStop : BOOL ;
  InSimulation : BOOL ;
  InNoSuspend : BOOL ;
  StStopped : BOOL ;
  StSuspend : BOOL ;
  StRunning : BOOL ;
  StFault : BOOL ;
  OutWarning : BOOL ;
  OutMonPressure : BOOL ;
  OutFaultRelevant : BOOL ;
  OutSuspendDelayRunning : BOOL ;
  OutSuspendDelayEnd : BOOL ;
  OutTargetReached : BOOL ;
  OutReleaseTrending : BOOL ;
  OutReleaseFeeding : BOOL ;	//Release to start of the suspend machines.
  InValueTarget : DINT ;	//[Pa] Target air pressure value
  InValueActual : REAL ;	//[Pa] Actual air pressure value
  InFUMaxFrequency : INT ;
  OutFUTargetFrequency : REAL ;
  OutTimeStarted : DINT ;
  OutTimeFaulted : DINT ;	//[s] Not errasable time "Faulted"
  OutCntStartup : DINT ;	//Not errasable counter of startup
  OutCntFault : DINT ;	//Not errasable counter of faults
  Fault : STRUCT
   Err00 : BOOL ;
   Err01 : BOOL ;
   Err02 : BOOL ;
   Err03 : BOOL ;
   Err04 : BOOL ;
   Err05 : BOOL ;
   Err06 : BOOL ;
   Err07 : BOOL ;
  END_STRUCT ;
  Par : STRUCT
   ParObjectNo : INT ;
   ParHornCode : INT ;	//Is used by horn module
   ParMsgType : INT ;
   ParLogOff : BOOL ;	//Report is off
   ParManual : BOOL ;	//Manual mode without interlocking
   ParSuspendTime : INT ;
   ParSuspendSpeed : INT ;
   ParManualSpeed : INT ;
   ParOverridePSTime : INT ;
   ParControllerTolerance : INT ;
   ParPressureTolerance : INT ;
  END_STRUCT ;
  PIDControl : FB 1541;
  SuspendDelay : FB 1706;
  ReleaseFeedDelay : FB 1706;
  PressureAlarmDelay : FB 1706;
  PressureRangeCheck : FB 1809;
  OutValueTarget : REAL ;
  PCRead : STRUCT
   ModeManual : BOOL ;
   TargetPressure : DINT ;
   Speed : INT ;
   Power : INT ;
   ActualPressure : DINT ;
  END_STRUCT ;
END_VAR
VAR_TEMP
  tmpInt : INT ;
  tmpBool : BOOL ;
  tmpLocal : BOOL ;
  tmpReport : BOOL ;
  tmpEnable : BOOL ;
  tmpFault : BOOL ;
  tmpLOGvalue : WORD ;	//LOG value
  tmpNewTargetValue : BOOL ;
END_VAR
BEGIN
NETWORK
TITLE = Methode: PID-Control
      AN    "GCS7_Gr_OutCallFast1";	//is set in time OB
      AN    "GCS7_Gr_OutCallFast2";	//is set in time OB
      AN    "GCS7_Gr_OutCallFast3";	//is set in time OB
      JC    oEnd;
// 
      L     DID [AR2,P#60.0];
      BLD   14;
      =     L 13.0;
      L     DINO;
      T     LW 11;
      CDB;
      OPN   DI [LW 11];
      TAR2  LD 7;
      CLR;
      =     DIX [AR2,P#58.2];
      SET;
      =     DIX [AR2,P#58.3];
      SET;
      =     DIX [AR2,P#58.4];
      CLR;
      =     DIX [AR2,P#58.5];
      CLR;
      =     DIX [AR2,P#58.6];
      CLR;
      =     DIX [AR2,P#58.7];
      L     L#0;
      T     DID [AR2,P#90.0];
      L     L#1184645120;
      T     DID [AR2,P#98.0];
      L     L#0;
      T     DID [AR2,P#102.0];
      +AR2  P#58.0;
      UC    FB 1541;
      LAR2  LD 7;
      CDB;
      BLD   15;
      BEU;
oEnd: NOP   0;
// 
NETWORK
TITLE = PC Control
      NOP   0;
//=== Test Object number =====================
      L     "SYS_DirectCtrlDB".PC.ObjectNo;	//PCControl.ObjectNo
      L     #Par.ParObjectNo;	//Input ObjectNo
      <>I;
      JC    Ctrl;
//=== Test OType      ========================
      L     1841;	//Input object type
      L     "SYS_DirectCtrlDB".PC.ObjectType;	//PCControl.ObjectType
      <>I;
      JC    Ctrl;
//=== Test Handshake =========================
      A     "SYS_DirectCtrlDB".PC.Hsk.FExamine;	// Handshake.FExamine
      JC    pExa;
      A     "SYS_DirectCtrlDB".PC.Hsk.FDefineCmd;	// Handshake.FDefineCmd
      JC    pCmd;
      A     "SYS_DirectCtrlDB".PC.Hsk.FDefinePara;	// Handshake.FDefinePara
      JC    pPar;
pIni: L     2;	// FcInit
      UC    "SYS_DirectCtrl";
      JU    Ctrl;
// Write parameter 
pPar: L     "SYS_DirectCtrlDB".PC.Value[11];
      T     #Par.ParSuspendTime;
      L     "SYS_DirectCtrlDB".PC.Value[12];
      T     #Par.ParSuspendSpeed;
      L     "SYS_DirectCtrlDB".PC.Value[13];
      T     #Par.ParManualSpeed;
      L     "SYS_DirectCtrlDB".PC.Value[14];
      T     #Par.ParOverridePSTime;
      L     "SYS_DirectCtrlDB".PC.Value[15];
      T     #Par.ParControllerTolerance;
      L     "SYS_DirectCtrlDB".PC.Value[16];
      T     #Par.ParPressureTolerance;
// Write new commands from PC to Interface object
pCmd: A     "SYS_DirectCtrlDB".PC.Cmd2[6];	// CmdFullLoadOn
      S     #InFullLoad;
      A     "SYS_DirectCtrlDB".PC.Cmd2[10];	// CmdNext
      S     #CmdNext;
      A     "SYS_DirectCtrlDB".PC.Cmd2[11];	// CmdFaultReset
      S     #CmdFaultReset;
      A     "SYS_DirectCtrlDB".PC.Cmd2[13];	// CmdManualOn
      S     #InManual;
      A     "SYS_DirectCtrlDB".PC.Cmd2[14];	// CmdReportOn
      S     #InReport;
      A     "SYS_DirectCtrlDB".PC.Cmd3[6];	// CmdFullLoadOff
      R     #InFullLoad;
      A     "SYS_DirectCtrlDB".PC.Cmd3[13];	// CmdManualOff
      R     #InManual;
      A     "SYS_DirectCtrlDB".PC.Cmd3[14];	// CmdReportOff
      R     #InReport;
//-----------------------------------------------------------
      JU    pIni;
pExa: L     #OutTimeStarted;	//[6.5]
      T     "SYS_DirectCtrlDB".PC.Value[7];	//[6.5]
      L     #OutTimeFaulted;	//[6.5]
      T     "SYS_DirectCtrlDB".PC.Value[8];	//[6.5]
      L     #OutCntStartup;	//[6.5]
      T     "SYS_DirectCtrlDB".PC.Value[9];	//[6.5]
      L     #OutCntFault;	//[6.5]
      T     "SYS_DirectCtrlDB".PC.Value[10];	//[6.5]
      L     #Par.ParSuspendTime;
      T     "SYS_DirectCtrlDB".PC.Value[11];
      L     #Par.ParSuspendSpeed;
      T     "SYS_DirectCtrlDB".PC.Value[12];
      L     #Par.ParManualSpeed;
      T     "SYS_DirectCtrlDB".PC.Value[13];
      L     #Par.ParOverridePSTime;
      T     "SYS_DirectCtrlDB".PC.Value[14];
      L     #Par.ParControllerTolerance;
      T     "SYS_DirectCtrlDB".PC.Value[15];
      L     #Par.ParPressureTolerance;
      T     "SYS_DirectCtrlDB".PC.Value[16];
//------------------------------------------
      TAR2;	// Address Dynamic datas
      T     "SYS_DirectCtrlDB".GC.InDynAddr;	// -->PCControl.GC.InDynAddr
      L     300;	// Length Dynamic datas
      T     "SYS_DirectCtrlDB".GC.InDynLen;	// -->PCControl.GC.InDynLen
      L     0;
      T     "SYS_DirectCtrlDB".GC.InParaAddr;	// -->PCControl.GC.InParaAddr
      T     "SYS_DirectCtrlDB".GC.InParaLen;	// -->PCControl.GC.InParaLen
      L     10;	// Revision
      T     "SYS_DirectCtrlDB".GC.Revision;	// 
      L     DINO;
      T     "SYS_DirectCtrlDB".GC.InDBNr;
      JU    pIni;
Ctrl: NOP   0;
NETWORK
TITLE =  All State Init
      NOP   0;
//===Clear tmp Variable, when nessecary
      CLR;
      =     #tmpBool;
//===Global Group Orders===
//      U     "SSW_Flag_GrOutManualOff"
//      R     #InManual
      AN    #InManual;
      A     #InLocal;
      =     #tmpLocal;
//Global FaultReset
      A     "GCS7_Gr_OutFaultReset";
      S     #CmdFaultReset;
//---Report is on---
      O     "GCS7_Gr_OutReportAll";
      O     #InReport;
      =     #tmpReport;
//---Enable / Automatic Interlocking Mode---
      A     #InEnable;
      AN    #InHWStop;
      AN    #InLocal;
      =     #tmpEnable;
//-Fault---
      O     #Fault.Err00;
      O     #Fault.Err01;
      O     #Fault.Err02;
      O     #Fault.Err03;
      O     #Fault.Err04;
      O     #Fault.Err05;
      O     #Fault.Err06;
      O     #Fault.Err07;
      =     #tmpFault;
//-Target value---
      L     #InValueTarget;
      L     DID [AR2,P#282.0];
      <>D;
      =     #tmpNewTargetValue;
      L     #InValueTarget;
      T     DID [AR2,P#282.0];
NETWORK
TITLE = CC: PID Controller configuration
// (network holds code this reader does not know; not shown)
// 
//-Enable controller---
// 
//-Manual mode---
// 
//- Target value---
// 
//-Target value manual mode---
// 
// 
// 
// 
//-Actual value---
// 
//-Dead band---
// 
//-Output value adaption---
NETWORK
TITLE = Timer control
      NOP   0;
// 
//-Suspend---
      AN    #tmpEnable;	//[1.1]
      O     #InNoSuspend;	//[1.1]
      =     DIX [AR2,P#184.0];	//[1.1]
// 
      BLD   14;
      =     L 13.0;
      L     DINO;
      T     LW 11;
      CDB;
      OPN   DI [LW 11];
      TAR2  LD 7;
      CLR;
      =     DIX [AR2,P#184.1];
      CLR;
// 
//-Pressure alarm---
      =     DIX [AR2,P#184.2];
      CLR;
      =     DIX [AR2,P#184.3];
      SET;
      =     DIX [AR2,P#184.4];
// 
      L     DBW [AR2,P#46.0];
      T     DIW [AR2,P#186.0];
      +AR2  P#184.0;
      UC    FB 1706;
      LAR2  LD 7;
      CDB;
      BLD   15;
      AN    #tmpNewTargetValue;
      AN    #InManual;
      AN    #InFullLoad;
// 
//-Release feeding---
      A     #InNoSuspend;
      =     DIX [AR2,P#240.0];
// 
      BLD   14;
      =     L 13.0;
// 
      L     DINO;
      T     LW 11;
      CDB;
      OPN   DI [LW 11];
      TAR2  LD 7;
      CLR;
      =     DIX [AR2,P#240.1];
      SET;
      =     DIX [AR2,P#240.2];
      CLR;
      =     DIX [AR2,P#240.3];
      SET;
      =     DIX [AR2,P#240.4];
      L     DBW [AR2,P#52.0];
      T     DIW [AR2,P#242.0];
      +AR2  P#240.0;
      UC    FB 1706;
      LAR2  LD 7;
      CDB;
      BLD   15;
      A     #OutTargetReached;
      S     DIX [AR2,P#212.0];
      AN    #InNoSuspend;
      R     DIX [AR2,P#212.0];
      BLD   14;
      =     L 13.0;
      L     DINO;
      T     LW 11;
      CDB;
      OPN   DI [LW 11];
      TAR2  LD 7;
      CLR;
      =     DIX [AR2,P#212.1];
      SET;
      =     DIX [AR2,P#212.2];
      CLR;
      =     DIX [AR2,P#212.3];
      SET;
      =     DIX [AR2,P#212.4];
      L     10;
      T     DIW [AR2,P#214.0];
      +AR2  P#212.0;
      UC    FB 1706;
      LAR2  LD 7;
      CDB;
      BLD   15;
NETWORK
TITLE = States
      A     #StStopped;	//===State machine===
      JC    S0;
      O     #StSuspend;
      JC    S1;
      A     #StRunning;
      JC    S3;
      A     #StFault;
      JC    S4;
      S     #StStopped;	//Initialise: goto StStopped
NETWORK
TITLE = StStopped
      NOP   0;
//==============================
// Any transition to StStopped
//==============================
xxS0: SET;
      S     #StStopped;
      JU    LOG1;
//==============================
//State
//==============================
//---Condition for StFault
S0:   A     #tmpFault;
      AN    #tmpLocal;
      JC    S0S4;
//---Condition for StRunning
      A     #tmpEnable;
      JC    S0S3;	//[1.1]
      JU    SAVE;
//[1.1]//---Transition -> StSuspend
//[1.1]S0S1: R     #StStopped
//[1.1]      SPA   xxS1
//---Transition -> StRunning            //[1.1]
S0S3: R     #StStopped;	//[1.1]
      JU    xxS3;	//[1.1]
//---Transition -> StFault
S0S4: R     #StStopped;
      JU    xxS4;
NETWORK
TITLE = StSuspend
      NOP   0;
//==============================
// Any transition to StSuspend
//==============================
xxS1: SET;
      S     #StSuspend;
      JU    LOG1;
//==============================
//State
//==============================
//---Condition for StFault
S1:   A     #tmpFault;
      AN    #tmpLocal;
      JC    S1S4;
//---Condition for StStopped
      AN    #tmpEnable;
      O     #tmpLocal;
      JC    S1S0;
//---Condition for StRunning
      A     #InNoSuspend;
      JC    S1S3;
      JU    SAVE;
//---Transition -> StStopped
S1S0: R     #StSuspend;
      JU    xxS0;
//---Transition -> StRunning
S1S3: R     #StSuspend;
      JU    xxS3;
//---Transition -> StFault
S1S4: R     #StSuspend;
      JU    xxS4;
NETWORK
TITLE = StRunning
      NOP   0;
//==============================
// Any transition to StRunning
//==============================
xxS3: SET;
      S     #StRunning;
      JU    LOG1;
//==============================
//State
//==============================
//---Condition for StFault
S3:   A     #tmpFault;
      AN    #tmpLocal;
      JC    S3S4;
//---Condition for StStopped
      AN    #tmpEnable;
      O     #tmpLocal;
      JC    S3S0;
//---Condition for StSuspend
      AN    DIX [AR2,P#188.0];
      JC    S3S1;
      JU    SAVE;
//---Transition -> StStopped
S3S0: R     #StRunning;
      JU    xxS0;
//---Transition -> StSuspend
S3S1: R     #StRunning;
      JU    xxS1;
//---Transition -> StFault
S3S4: R     #StRunning;
      JU    xxS4;
NETWORK
TITLE =  StFault
      NOP   0;
//==============================
// Any transiton to Fault  
//==============================
// Maintanance Counter Faults
xxS4: A     #StFault;
      JC    S4T2;
      L     #OutCntFault;
      +     L#1;
      T     #OutCntFault;
S4T2: SET;
      S     #StFault;
      S     "GCS7_Gr_InFault";
      CALL  "SYS_Horn_Code" (
           FcCode                   := 1,
           ParObjectType            := 1841,
           ParObjectNo              := #Par.ParObjectNo,
           ParHornCode              := #Par.ParHornCode);
S4S4: JU    LOG4;
//==============================
//State
//==============================
// Maintanance Counter Fault Time
S4:   AN    "GCS7_Gr_OutTick1s";	// Increment all s
      JC    S4MT;
      L     #OutTimeFaulted;
      +     L#1;
      T     #OutTimeFaulted;
//===logic
S4MT: AN    #CmdFaultReset;	//---Condition for StFault
      AN    #tmpLocal;
      JC    SAVE;
//---Condition for StFault with LOG
      A     #tmpFault;
      AN    #tmpLocal;
      JC    S4S4;
      R     #StFault;	//---Transition -> StStopping
      S     #StStopped;
      JU    LOG9;
NETWORK
TITLE = LOG Message
//LOG transition to an other state
LOG1: AN    #tmpReport;	// ReportAll
      JC    SAV2;
      A     #StRunning;
      L     B#(4, 2);	// MessageClass Info Running
      JC    LOG;
      A     #StSuspend;
      L     B#(4, 1);	// MessageClass Info Suspend
      JC    LOG;
      A     #StStopped;
      L     B#(4, 0);	// MessageClass Info Stopped
      JC    LOG;
      JU    SAV2;
//LOG transition to fault
LOG4: A     #Fault.Err01;
      L     B#(1, 11);	// MessageClass Error ErrX
      JC    LOG;
      JU    SAV2;
      CLR;
      L     B#(4, 15);	// MessageClass Info 
      JC    LOG;
      JU    SAV2;
//Log fault cancelled
LOG9: L     B#(3, 9);	// MessageClass Operater "fault cancelled"
LOG:  A     #Par.ParLogOff;	//---Set LOG Message
      JC    SAV2;
      T     #tmpLOGvalue;
// 
      CALL  "GCS7_LogConvert" (
           ObjectNo                 := #Par.ParObjectNo,
           MsgType                  := #Par.ParMsgType,
           ClassMsgTxt              := #tmpLOGvalue,
           OType                    := 1841);
SAV2: NOP   0;
NETWORK
TITLE = State Code
SAVE: NOP   0;
//--Stopped, Substate ---
      A     #StStopped;
      L     1;	// Code: stopped
      JC    STC9;
//--------------------
      A     #InFullLoad;
      L     5;	// Code: full load 
      JC    STC9;
//--------------------
      A     #StSuspend;
      L     2;	// Code: suspend
      JC    STC9;
//--------------------
      A     #StRunning;
      L     4;	// Code: running 
      JC    STC9;
      L     32;	// Code: fault
//----------------------
STC9: L     #StCode;	// Old state code
      TAK;
      T     #StCode;	// Save state code
      <>I;
      L     3;	// Load code for CBit methode
      CC    "SYS_CBitCtrl";
NETWORK
TITLE = Out signals
      NOP   0;
//-Warning---
      A     #InWarning;
      A     #StFault;
      =     #OutWarning;
// 
//-Pressure monitoring---
      AN    #InManual;
      AN    #InFullLoad;
      AN    #InNoPressureAlarm;
      A     DIX [AR2,P#244.0];
      =     #OutMonPressure;
// 
//-Relevant fault---
      AN    M 11.7;
      ON    #InLocal;
      A     #StFault;
      AN    #InWarning;
      =     #OutFaultRelevant;
// 
//-Timer states---
      AN    DIX [AR2,P#184.0];
      A     DIX [AR2,P#188.0];
      =     #OutSuspendDelayRunning;
      AN    DIX [AR2,P#188.0];
      =     #OutSuspendDelayEnd;
// 
//-Target reached---
      L     #InValueTarget;
      DTR;
      T     DID [AR2,P#268.0];
// 
      L     #Par.ParPressureTolerance;
      ITD;
      DTR;
      T     DID [AR2,P#276.0];
// 
      BLD   14;
      =     L 13.0;
      L     DINO;
      T     LW 11;
      CDB;
      OPN   DI [LW 11];
      TAR2  LD 7;
      L     DBD [AR2,P#10.0];
      T     DID [AR2,P#272.0];
      +AR2  P#268.0;
// 
//-Release trending---
      UC    FB 1809;
      LAR2  LD 7;
// 
//-Frequency convertor target value---
      A     DIX [AR2,P#280.1];
      =     DBX [AR2,P#4.7];
// 
//-Release suspend machines---
      CDB;
      BLD   15;
      A     DIX [AR2,P#188.0];
      =     #OutReleaseTrending;
      L     DID [AR2,P#130.0];
      T     #OutFUTargetFrequency;
      O     DIX [AR2,P#216.0];
      O     #InManual;
      =     #OutReleaseFeeding;
NETWORK
TITLE = PCRead
      A     #InManual;
      =     DIX [AR2,P#286.0];
// 
      L     #InValueTarget;
      T     DID [AR2,P#288.0];
// 
// Handled in group      T     #PCRead.Speed
// Handled in group      T     #PCRead.Power
// 
      L     #InValueActual;
      RND;
      T     DID [AR2,P#296.0];
NETWORK
TITLE = Global End
      NOP   0;
//-Clear all commands---
      CLR;
      =     #CmdNext;
      =     #CmdFaultReset;
//--Output for group 
      A     M 11.7;
      A     #InLocal;
      A     #InManual;
//      O     #InForce
      JC    ENJ2;
      A     #InHWStop;
      S     "GCS7_Gr_InHWStop";
ENJ2: A     #InManual;
      S     "GCS7_Gr_InManual";
NETWORK
TITLE = End of block
      BE;
END_FUNCTION_BLOCK

FUNCTION_BLOCK "SSW_EL_ASI_Fct"	// FB 899
TITLE = ASI Master
//
//COPYRIGHT:    (C) 1996  BUHLER AG, CH-9240 UZWIL, SWITZERLAND
//
//PRODUCT:      GCS7R2
//
//TITLE:        SSW_ASI_Wago_Fct
//
//REVISION:     20
//-------------------------------------------------------------------------
//
//IDENT:        AUTHOR:             DEPT:                       DATE:
//FB899.1.1     Ph. Engler          GP92                        17-Apr-2009
//              LOG: Text numbers changed
//FB899.1.0     A.Egli              BASE                        03-Mar-2009
//              1st Release in S7
//
//-------------------------------------------------------------------------
//
//PURPOSE:      MANUAL : see [SSW-EL-ASI_MAN_en]
//
//RESTRICTIONS: S7
//
//-------------------------------------------------------------------------
//=======================================================
//Log Message: 
//------------------------------------------------------
//11  fault ASI-Master
//12  fault ASI-Slave
//
//=======================================================
//StCode:  State               
//------------------------------------------------------
// 0 StNotUsed   : Slave not used
// 2 StOk        : ok
//32 StFault
//33 StFault.DPMaster  
//34 StFault.ASIMaster            
//35 StFault.CfgDiff             (Slave only)
//36 StFault.PeripheralFault     (Slave only)
//37 StFault.Corrupted           (Slave only) 
//38 StFault.Overflow            (Master only) 
//39 StFault.ASIInactive         (Master only) 
//40 StFault.ErrPower            (Master only) 
//41 StFault.ErrMapping          (Master only) 
//42 StFault.ErrGeneral          (Master only) 
//
//
AUTHOR : EA
FAMILY : GCS7LL
NAME : EL_ASI
VERSION : 1.1
VAR
  StCode : INT ;	//Element state code
  InDPFault : BOOL ;	//DP-Fault is detected, no fault
  InLogOff : BOOL ;	//No Log Message
  InHornOff : BOOL ;	//No Alarm Horn
  CmdFaultReset : BOOL ;	//Command to reset fault
  Spare3 : BYTE ;
  OutDPFault : BOOL ;
  OutFaultRelevant : BOOL ;	//Relevant Fault of ASIMaster
  OutMsgDone : BOOL ;	//LOG Message Done
  Spare43 : BOOL ;
  Spare44 : BOOL ;
  Spare45 : BOOL ;
  Spare46 : BOOL ;
  Spare47 : BOOL ;
  Spare51 : BOOL ;
  Spare52 : BOOL ;
  StOk : BOOL ;	//Element is stopped
  Spare53 : BOOL ;
  StFault : BOOL ;	//Element has a fault
  Fault : STRUCT
   DPMaster : BOOL ;	//DPMaster not active
   ASIMaster : BOOL ;	//ASI Master not response
   Overflow : BOOL ;	//1=data not complet (timing)
   ASIInactive : BOOL ;	//1=ASI Interface inactive / 0= Active
   ErrPower : BOOL ;	//1=Power fault/24V
   ErrMapping : BOOL ;	//1=data not complett, mapping
   CfgMode : BOOL ;	//1=Configuration mode / 0= Protected
   ErrGeneral : BOOL ;	//1=Any fault
  END_STRUCT ;
  OutAlarmNoLog : INT ;	//Last textnumber send to log
  OutTimeStarted : DINT ;	//not used
  OutTimeFaulted : DINT ;	//not used
  OutCntStartup : DINT ;	//not used
  OutCntFault : DINT ;	//not used
  Slaves_Detected : STRUCT 	//1= Detected Slaves A (Read with 0x46)
   A : ARRAY  [0 .. 31 ] OF BOOL ;
   B : ARRAY  [0 .. 31 ] OF BOOL ;
  END_STRUCT ;
  Slaves_CfgDiff : STRUCT 	//1= Slaves A with configuartion diff.(Read with 0x57)
   A : ARRAY  [0 .. 31 ] OF BOOL ;
   B : ARRAY  [0 .. 31 ] OF BOOL ;
  END_STRUCT ;
  Slaves_PeripheralFault : STRUCT 	//1= Slaves A peripheral failure (Read with 0x3E)
   A : ARRAY  [0 .. 31 ] OF BOOL ;
   B : ARRAY  [0 .. 31 ] OF BOOL ;
  END_STRUCT ;
  Slaves_Corrupted : STRUCT 	//1= Corrupped Slaves A (Read with 0x6C)
   A : ARRAY  [0 .. 31 ] OF BOOL ;
   B : ARRAY  [0 .. 31 ] OF BOOL ;
  END_STRUCT ;
  Slaves_Faulted : STRUCT 	//1= Faulted Slaves A (Summery state)
   A : ARRAY  [0 .. 31 ] OF BOOL ;
   B : ARRAY  [0 .. 31 ] OF BOOL ;
  END_STRUCT ;
  tmpSlave : UDT 28995;
  Slaves : STRUCT
   A : ARRAY  [1 .. 31 ] OF UDT 28995;
   B : ARRAY  [0 .. 31 ] OF UDT 28995;
  END_STRUCT ;
  Com : STRUCT
   IdxSlave : INT ;	//Current Slave
   OutResult : INT ;	//Result Value Mailbox communication
  END_STRUCT ;
  Snd : STRUCT
   Control : STRUCT
    Cmd0 : BOOL ;
    Cmd1 : BOOL ;
    Cmd2 : BOOL ;
    Cmd3 : BOOL ;
    Cmd4 : BOOL ;
    Mbx : BOOL ;	//1=Mailbox on
    R_W : BOOL ;	//1=Write , 0=Read
    RegisterCom : BOOL ;	//1=Register communication
    Internal : BYTE ;
   END_STRUCT ;
   Mailbox : STRUCT
    Opcode : BYTE ;
    spare20 : BOOL ;
    spare21 : BOOL ;
    spare22 : BOOL ;
    spare23 : BOOL ;
    spare24 : BOOL ;
    B_A : BOOL ;	//1=B / 0=A
    Order : BOOL ;	//1=Parameter bytes order invers
    Toggle : BOOL ;	//Bit must toogle
    Slave : BYTE ;
    Value1High : BYTE ;
    Value1Low : BYTE ;
    Value2High : BYTE ;
    Value2Low : BYTE ;
    Value3High : BYTE ;
    Value3Low : BYTE ;
    Value4High : BYTE ;
    Value4Low : BYTE ;
    spare : BYTE ;
   END_STRUCT ;
   ProcessData : ARRAY  [1 .. 288 ] OF BOOL ;
  END_STRUCT ;
  Rcv : STRUCT
   Status : STRUCT
    Overflow : BOOL ;	//1=data not complett timing
    ASIInactive : BOOL ;	//1=ASI Interface inactive / 0= Active
    ErrPower : BOOL ;	//1=Power fault/24V
    ErrMapping : BOOL ;	//1=data not complett, mapping
    CfgMode : BOOL ;	//1=Configuration mode / 0= Protected
    MailBox : BOOL ;	//1=Mailbox is fade in
    ErrGeneral : BOOL ;	//1=Any fault
    AckProcessData : BOOL ;	//1=Acknowledge process data
    Internal : BYTE ;
   END_STRUCT ;
   Mailbox : STRUCT
    Opcode : BYTE ;	//Copy of Snd.Mailbox.Opcode
    Result0 : BOOL ;
    Result1 : BOOL ;
    Result2 : BOOL ;
    Result3 : BOOL ;
    Result4 : BOOL ;
    Result5 : BOOL ;	//1=B / 0=A
    Result7 : BOOL ;	//1=Parameter bytes order invers
    Toggle : BOOL ;	//Bit must toogle
    ValueAB : DWORD ;
    ValueBA : DWORD ;
    spare : WORD ;
   END_STRUCT ;
   ProcessData : ARRAY  [1 .. 288 ] OF BOOL ;
  END_STRUCT ;
  Par : STRUCT
   ParObjectNo : INT ;	//Is used for communication with PC, e.g. for message
   ParMsgType : INT ;
   ParHornCode : INT ;	//Is used by horn module
   ParLogOff : BOOL ;	//Report is off
   ParDPNode : INT ;
   ParASIMasterIdx : INT  := 1;	//Index of ASI Master
   ParIOByteNo : INT  := 100;
   ParLenMailbox : INT  := 12;
   ParMonTime : INT  := 10;	//[0.1 s] Maximum reposnse time Slave
   OutMonTime : INT ;	//[0.1 s] Maximum reposnse time
  END_STRUCT ;
END_VAR
VAR_TEMP
  tmpLOGvalue : WORD ;	//LOG value
  tmpReport : BOOL ;	//Global LOG all
  tmpAddrIO : DWORD ;
  tmpMailboxLong : BOOL ;
  tmpLenSlaveData : DINT ;	//Lenght as Bits
  tmpObjectNo : DINT ;
  tmpAddr : DINT ;	//Address Current Slave in Array
  tmpIdx : INT ;
  tmpUsed : BOOL ;
  tmpDPFault : BOOL ;
  tmpRelavantFaultSlaves : BOOL ;
  tmpPar1 : WORD ;
  tmpPar2 : WORD ;
  tmpPar3 : WORD ;
  tmpHeader : WORD ;
END_VAR
BEGIN
NETWORK
TITLE = PC Control
//=== Test Object number =====================
      L     "SYS_DirectCtrlDB".PC.ObjectNo;	//PCControl.ObjectNo
      L     #Par.ParObjectNo;	//Input ObjectNo
      <>I;
      JC    Ctrl;
//=== Test OType      ========================
      L     1899;	//Input object type
      L     "SYS_DirectCtrlDB".PC.ObjectType;	//PCControl.ObjectType
      <>I;
      JC    Ctrl;
//=== Test Handshake =========================
      A     "SYS_DirectCtrlDB".PC.Hsk.FExamine;	// Handshake.FExamine
      JC    pExa;
      A     "SYS_DirectCtrlDB".PC.Hsk.FDefineCmd;	// Handshake.FDefineCmd
      JC    pCmd;
      A     "SYS_DirectCtrlDB".PC.Hsk.FDefinePara;	// Handshake.FDefinePara
      JC    pPar;
pIni: L     2;	// FcInit
      UC    "SYS_DirectCtrl";
      JU    Ctrl;
// Write parameter 
pPar: LAR1  P#DBX 58.0;
      L     P##Par;
      L     DW#16#FFFFF;
      AD;
      +AR1;
// Write new commands from PC to Interface object
pCmd: A     "SYS_DirectCtrlDB".PC.Cmd1[11];	// CmdFaultReset
      S     #CmdFaultReset;
      A     "SYS_DirectCtrlDB".PC.Cmd1[14];	// CmdReportOn
      R     #InLogOff;
      A     "SYS_DirectCtrlDB".PC.Cmd2[14];	// CmdReportOff
      S     #InLogOff;
      A     "SYS_DirectCtrlDB".PC.Cmd1[15];	// CmdHornOn
      R     #InHornOff;
      A     "SYS_DirectCtrlDB".PC.Cmd2[15];	// CmdHornOff
      S     #InHornOff;
      JU    pIni;
pExa: TAR2;	// Address Dynamic datas
      T     "SYS_DirectCtrlDB".GC.InDynAddr;	// -->PCControl.GC.InDynAddr
      L     20;	// Length Dynamic datas
      T     "SYS_DirectCtrlDB".GC.InDynLen;	// -->PCControl.GC.InDynLen
      L     0;
      T     "SYS_DirectCtrlDB".GC.InParaAddr;	// -->PCControl.GC.InParaAddr
      T     "SYS_DirectCtrlDB".GC.InParaLen;	// -->PCControl.GC.InParaLen
      L     1;	// Code FcExamine
      UC    "SYS_DirectCtrl";
      L     20;	//Revision
      T     "SYS_DirectCtrlDB".GC.Revision;
Ctrl: NOP   0;
NETWORK
TITLE = DPFault
      A     #InDPFault;
      =     #OutDPFault;
NETWORK
TITLE = Init
      L     #Par.ParLenMailbox;
      L     10;
      >=I;
      =     #tmpMailboxLong;
      L     P##Slaves;
      L     P##tmpSlave;
      -D;
      T     #tmpLenSlaveData;
NETWORK
TITLE = Input Data Status + Mailbox
      L     #Par.ParIOByteNo;
      SLD   3;
      T     #tmpAddrIO;
//Copy Status
      LAR1  #tmpAddrIO;
      L     IW [AR1,P#0.0];
      LAR1  P##Rcv;
      T     DIW [AR1,P#0.0];
//Copy Mailbox
      LAR1  #tmpAddrIO;
      L     IW [AR1,P#2.0];
      LAR1  P##Rcv;
      T     DIW [AR1,P#2.0];
//Copy Mailbox
      LAR1  #tmpAddrIO;
      L     ID [AR1,P#4.0];
      T     #Rcv.Mailbox.ValueAB;
      AN    #tmpMailboxLong;
      JC    RDJ0;
//Copy Mailbox
      LAR1  #tmpAddrIO;
      L     ID [AR1,P#8.0];
      T     #Rcv.Mailbox.ValueBA;
RDJ0: NOP   0;
NETWORK
TITLE = Mailbox: Answer
      L     #Snd.Mailbox.Opcode;
      L     #Rcv.Mailbox.Opcode;
      ==I;
      A(;
      A     #Snd.Mailbox.Toggle;
      A     #Rcv.Mailbox.Toggle;
      O;
      AN    #Snd.Mailbox.Toggle;
      AN    #Rcv.Mailbox.Toggle;
      );
      JC    MTOK;
      AN    "GCS7_Gr_OutTick200ms";	// Decrement all 200ms
      JC    MTJ0;
      L     #Par.OutMonTime;
      +     -2;
      T     #Par.OutMonTime;
      L     0;
      >=I;
      JC    MTJ0;
//=========================================================
//--Timeout Response ----
//=========================================================
      S     #Fault.ASIMaster;
      L     #Par.ParMonTime;
      T     #Par.OutMonTime;
      L     W#16#46;	// Read Opcode Detected Slave
      JU    MNXA;	//-->Send Next Command  
//=========================================================
//--Timeout Ok ----
//=========================================================
MTOK: R     #Fault.ASIMaster;
      L     #Par.ParMonTime;
      T     #Par.OutMonTime;
MTJ0: NOP   0;
NETWORK
TITLE = Mailbox: Check Togle Bit
      X     #Snd.Mailbox.Toggle;
      X     #Rcv.Mailbox.Toggle;
      O(;
      L     #Snd.Mailbox.Opcode;
      L     #Rcv.Mailbox.Opcode;
      <>I;
      );
      JC    MOUT;
      LAR1  P##Rcv;
      L     DIB [AR1,P#3.0];	//Rcv.Mailbox.Result
      L     2#1111111;
      AW;
      T     #Com.OutResult;
NETWORK
TITLE = Mailbox: Detected Slaves Ox46
      NOP   0;
      L     #Rcv.Mailbox.Opcode;
      L     W#16#46;	// Opcode Detected Slaves
      <>I;
      JC    M57;
      AN    #tmpMailboxLong;
      JC    M46S;	//Short Mailbox
//----------------------------------------------------
//--Long Mailbox
      LAR1  P##Slaves_Detected;
      L     #Rcv.Mailbox.ValueAB;
      T     DID [AR1,P#0.0];
      L     #Rcv.Mailbox.ValueBA;
      T     DID [AR1,P#4.0];
//Next Command
      L     W#16#57;	// Opcode Configuration Difference
      JU    MNXA;	//-->Send Next Command
//----------------------------------------------------
//--Short Mailbox
M46S: A     #Snd.Mailbox.B_A;
      JC    M46B;
      LAR1  P##Slaves_Detected;
      L     #Rcv.Mailbox.ValueAB;
      T     DID [AR1,P#0.0];
      L     #Rcv.Mailbox.Opcode;	// Read Slaves B
      JU    MNXB;	//-->Send Next Command
M46B: LAR1  P##Slaves_Detected;
      L     #Rcv.Mailbox.ValueAB;
      T     DID [AR1,P#4.0];
      L     W#16#57;	// Opcode Configuration Difference
      JU    MNXA;	//-->Send Next Command 
NETWORK
TITLE = Mailbox: Configuration DIfferent Ox57
      NOP   0;
M57:  L     #Rcv.Mailbox.Opcode;
      L     W#16#57;	// Opcode Detected Slaves
      <>I;
      JC    M3E;
      LAR1  P##Slaves_CfgDiff;
      AN    #tmpMailboxLong;
      JC    M57S;	//Short Mailbox
//----------------------------------------------------
//--Long Mailbox
      L     #Rcv.Mailbox.ValueAB;
      T     DID [AR1,P#0.0];
      L     #Rcv.Mailbox.ValueBA;
      T     DID [AR1,P#4.0];
//Next Command
      L     W#16#3E;	// Opcode Peripheral Failure
      JU    MNXA;	//-->Send Next Command
//----------------------------------------------------
//--Short Mailbox
M57S: A     #Snd.Mailbox.B_A;
      JC    M57B;
      L     #Rcv.Mailbox.ValueAB;
      T     DID [AR1,P#0.0];
      L     #Rcv.Mailbox.Opcode;	// Read Slaves B
      JU    MNXB;	//-->Send Next Command
M57B: L     #Rcv.Mailbox.ValueAB;
      T     DID [AR1,P#4.0];
      L     W#16#3E;	// Opcode Peripheral Failure
      JU    MNXA;	//-->Send Next Command 
NETWORK
TITLE = Mailbox: Configuration Pheriperal Failure Ox3E
      NOP   0;
M3E:  L     #Rcv.Mailbox.Opcode;
      L     W#16#3E;	// Opcode Pheriperal Failure
      <>I;
      JC    M6C;
      LAR1  P##Slaves_PeripheralFault;
      AN    #tmpMailboxLong;
      JC    M3ES;	//Short Mailbox
//----------------------------------------------------
//--Long Mailbox
      L     #Rcv.Mailbox.ValueAB;
      T     DID [AR1,P#0.0];
      L     #Rcv.Mailbox.ValueBA;
      T     DID [AR1,P#4.0];
//Next Command
      L     W#16#6C;	// Opcode Corrupted Slaves
      JU    MNXA;	//-->Send Next Command
//----------------------------------------------------
//--Short Mailbox
M3ES: A     #Snd.Mailbox.B_A;
      JC    M3EB;
      L     #Rcv.Mailbox.ValueAB;
      T     DID [AR1,P#0.0];
      L     #Rcv.Mailbox.Opcode;	// Read Slaves B
      JU    MNXB;	//-->Send Next Command
M3EB: L     #Rcv.Mailbox.ValueAB;
      T     DID [AR1,P#4.0];
      L     W#16#6C;	// Opcode Corrupted Slaves
      JU    MNXA;	//-->Send Next Command 
NETWORK
TITLE = Mailbox: Corrupted Slaves Ox6C
      NOP   0;
M6C:  L     #Rcv.Mailbox.Opcode;
      L     W#16#6C;	// Opcode Corrupted Slaves
      <>I;
      JC    M50;
      LAR1  P##Slaves_Corrupted;
      AN    #tmpMailboxLong;
      JC    M6CS;	//Short Mailbox
//----------------------------------------------------
//--Long Mailbox
      L     #Rcv.Mailbox.ValueAB;
      T     DID [AR1,P#0.0];
      L     #Rcv.Mailbox.ValueBA;
      T     DID [AR1,P#4.0];
//Next Command
      JU    M50I;	//-->Send Next Command
//----------------------------------------------------
//--Short Mailbox
M6CS: A     #Snd.Mailbox.B_A;
      JC    M6CB;
      L     #Rcv.Mailbox.ValueAB;
      T     DID [AR1,P#0.0];
      L     #Rcv.Mailbox.Opcode;	// Read Slaves B
      JU    MNXB;	//-->Send Next Command
M6CB: L     #Rcv.Mailbox.ValueAB;
      T     DID [AR1,P#4.0];
      JU    M50I;	//-->Send Next Command 
NETWORK
TITLE = Mailbox: Read Slaves Channel Ox50
      NOP   0;
//===========================================
//Init Reading Analog Values
M50I: L     0;
      T     #Com.IdxSlave;
      JU    M50X;
//===========================================
M50:  L     #Rcv.Mailbox.Opcode;
      L     W#16#50;	// Opcode Read Slave In Data Channel 1 to 4
      <>I;
      JC    M51;
      L     31;
      L     #Com.IdxSlave;
      <I;
      JC    M50X;
      L     1;
      L     #Com.IdxSlave;
      >I;
      JC    M50X;
      +     -1;
      T     #tmpIdx;
      L     #tmpLenSlaveData;
      *D;
      L     P##Slaves;
      +D;
      T     #tmpAddr;
//Copy Data from  SlavesA[x] to tmpSlave
      LAR1  #tmpAddr;
      L     DID [AR1,P#0.0];
      LAR1  P##tmpSlave;
      T     DID [AR1,P#0.0];
      LAR1  #tmpAddr;
      L     DID [AR1,P#4.0];
      LAR1  P##tmpSlave;
      T     DID [AR1,P#4.0];
      LAR1  #tmpAddr;
      L     DID [AR1,P#8.0];
      LAR1  P##tmpSlave;
      T     DID [AR1,P#8.0];
      LAR1  #tmpAddr;
      L     DID [AR1,P#12.0];
      LAR1  P##tmpSlave;
      T     DID [AR1,P#12.0];
//Read Values from Mailbox
      L     #Com.OutResult;
      T     #tmpSlave.OutResult;
      L     #Rcv.Mailbox.ValueAB;
      T     #tmpSlave.Ch2;
      SRD   16;
      T     #tmpSlave.Ch1;
      AN    #tmpMailboxLong;
      JC    M50S;	//--> Save Data
      L     #Rcv.Mailbox.ValueBA;
      T     #tmpSlave.Ch4;
      SRD   16;
      T     #tmpSlave.Ch3;
//Copy Data from tmpSlave of SlavesA[x]
M50S: LAR1  P##tmpSlave;
      L     DID [AR1,P#0.0];
      LAR1  #tmpAddr;
      T     DID [AR1,P#0.0];
      LAR1  P##tmpSlave;
      L     DID [AR1,P#4.0];
      LAR1  #tmpAddr;
      T     DID [AR1,P#4.0];
      LAR1  P##tmpSlave;
      L     DID [AR1,P#8.0];
      LAR1  #tmpAddr;
      T     DID [AR1,P#8.0];
      LAR1  P##tmpSlave;
      L     DID [AR1,P#12.0];
      LAR1  #tmpAddr;
      T     DID [AR1,P#12.0];
//------------------------------------------------------------------
//Loop Slave
//------------------------------------------------------------------
M50X: L     #Com.IdxSlave;
      +     1;
      T     #Com.IdxSlave;
      L     31;
      >I;
      JC    M51I;
      L     #Com.IdxSlave;
      +     -1;
      L     #tmpLenSlaveData;
      *D;
      L     P##Slaves;
      +D;
      T     #tmpAddr;
//Copy Data of SlavesA[x] to tmpSlave
      LAR1  #tmpAddr;
      L     DID [AR1,P#0.0];
      LAR1  P##tmpSlave;
      T     DID [AR1,P#0.0];
      AN    #tmpSlave.Par.ParAI;
      JC    M50X;
//==================================
//Prepare Mailbox Send
//==================================
      L     #Com.IdxSlave;
      T     #Snd.Mailbox.Slave;	//Enter Slave address
      L     W#16#50;	// Opcode Read Slave In Data Channel 1 to 4
      T     #Snd.Mailbox.Opcode;
      SET;
      R     #Snd.Mailbox.B_A;
      AN    #Rcv.Mailbox.Toggle;
      =     #Snd.Mailbox.Toggle;
      JU    MOUT;
NETWORK
TITLE = Mailbox: Write Slaves Channel Ox51
      NOP   0;
//===========================================
//Init Reading Analog Values
M51I: L     0;
      T     #Com.IdxSlave;
      JU    M51X;
//===========================================
M51:  L     #Rcv.Mailbox.Opcode;
      L     W#16#51;	// Opcode Write Slave Out Data Channel 1 to 4
      <>I;
      JC    MEND;	//MEND
      L     31;
      L     #Com.IdxSlave;
      <I;
      JC    M51X;
      L     1;
      L     #Com.IdxSlave;
      >I;
      JC    M51X;
      +     -1;
      T     #tmpIdx;
      L     #tmpLenSlaveData;
      *D;
      L     P##Slaves;
      +D;
      T     #tmpAddr;
//Copy Data from  SlavesA[x] to tmpSlave
      LAR1  #tmpAddr;
      L     DID [AR1,P#0.0];
      LAR1  P##tmpSlave;
      T     DID [AR1,P#0.0];
      LAR1  #tmpAddr;
      L     DID [AR1,P#4.0];
      LAR1  P##tmpSlave;
      T     DID [AR1,P#4.0];
      LAR1  #tmpAddr;
      L     DID [AR1,P#8.0];
      LAR1  P##tmpSlave;
      T     DID [AR1,P#8.0];
      LAR1  #tmpAddr;
      L     DID [AR1,P#12.0];
      LAR1  P##tmpSlave;
      T     DID [AR1,P#12.0];
//Read Values from Mailbox
      L     #Com.OutResult;
      T     #tmpSlave.OutResult;
//Copy Data from tmpSlave of SlavesA[x]
      LAR1  P##tmpSlave;
      L     DID [AR1,P#0.0];
      LAR1  #tmpAddr;
      T     DID [AR1,P#0.0];
      LAR1  P##tmpSlave;
      L     DID [AR1,P#4.0];
      LAR1  #tmpAddr;
      T     DID [AR1,P#4.0];
      LAR1  P##tmpSlave;
      L     DID [AR1,P#8.0];
      LAR1  #tmpAddr;
      T     DID [AR1,P#8.0];
      LAR1  P##tmpSlave;
      L     DID [AR1,P#12.0];
      LAR1  #tmpAddr;
      T     DID [AR1,P#12.0];
//------------------------------------------------------------------
//Loop Slave
//------------------------------------------------------------------
M51X: L     #Com.IdxSlave;
      +     1;
      T     #Com.IdxSlave;
      L     31;
      >I;
      JC    MEND;	//---> Start Sequence
      L     #Com.IdxSlave;
      +     -1;
      L     #tmpLenSlaveData;
      *D;
      L     P##Slaves;
      +D;
      T     #tmpAddr;
//Copy Data of SlavesA[x] to tmpSlave
      LAR1  #tmpAddr;
      L     DID [AR1,P#0.0];
      LAR1  P##tmpSlave;
      T     DID [AR1,P#0.0];
      AN    #tmpSlave.Par.ParAO;
      JC    M51X;
      LAR1  #tmpAddr;
      L     DID [AR1,P#4.0];
      LAR1  P##tmpSlave;
      T     DID [AR1,P#4.0];
      LAR1  #tmpAddr;
      L     DID [AR1,P#8.0];
      LAR1  P##tmpSlave;
      T     DID [AR1,P#8.0];
      LAR1  #tmpAddr;
      L     DID [AR1,P#12.0];
      LAR1  P##tmpSlave;
      T     DID [AR1,P#10.0];
//==================================
//Prepare Mailbox Send
//==================================
      L     #Com.IdxSlave;
      T     #Snd.Mailbox.Slave;	//Enter Slave address
      LAR1  P##Snd;
      +AR1  P#5.0;
      L     #tmpSlave.Ch1;
      T     DIW [AR1,P#0.0];
      L     #tmpSlave.Ch2;
      T     DIW [AR1,P#2.0];
      L     #tmpSlave.Ch3;
      T     DIW [AR1,P#4.0];
      L     #tmpSlave.Ch4;
      T     DIW [AR1,P#6.0];
      L     W#16#51;	// Opcode Write Slave In Data Channel 1 to 4
      T     #Snd.Mailbox.Opcode;
      SET;
      R     #Snd.Mailbox.B_A;
      AN    #Rcv.Mailbox.Toggle;
      =     #Snd.Mailbox.Toggle;
      JU    MOUT;
NETWORK
TITLE = Mailbox: Else 
MEND: L     W#16#46;	// Opcode Detected Slave
      JU    MNXA;	//-->Send Next Command  
NETWORK
TITLE = Mailbox: Enter Next command
//--------------------------------------
//Send Next Command Order A/B
//--------------------------------------
MNXA: T     #Snd.Mailbox.Opcode;
      SET;
      R     #Snd.Mailbox.B_A;
      JU    MNX;
//--------------------------------------
//Send Next Command Order B/A
//--------------------------------------
MNXB: T     #Snd.Mailbox.Opcode;
      SET;
      S     #Snd.Mailbox.B_A;
MNX:  AN    #Rcv.Mailbox.Toggle;
      =     #Snd.Mailbox.Toggle;
      L     0;
      T     #Snd.Mailbox.Slave;
      T     #Snd.Mailbox.Value1High;
      T     #Snd.Mailbox.Value1Low;
      T     #Snd.Mailbox.Value2High;
      T     #Snd.Mailbox.Value2Low;
      T     #Snd.Mailbox.Value3High;
      T     #Snd.Mailbox.Value3Low;
      T     #Snd.Mailbox.Value4High;
      T     #Snd.Mailbox.Value4Low;
MOUT: NOP   0;
NETWORK
TITLE = Mailbox Write to Output
//Copy Mailbox
      LAR1  P##Snd;
      L     DID [AR1,P#2.0];
      LAR1  #tmpAddrIO;
      T     QD [AR1,P#2.0];
      LAR1  P##Snd;
      L     DID [AR1,P#6.0];
      LAR1  #tmpAddrIO;
      T     QD [AR1,P#6.0];
      AN    #tmpMailboxLong;
      JC    MWJ0;
      LAR1  P##Snd;
      L     DID [AR1,P#10.0];
      LAR1  #tmpAddrIO;
      T     QD [AR1,P#10.0];
      LAR1  P##Snd;
      L     DIW [AR1,P#14.0];
      LAR1  #tmpAddrIO;
      T     QW [AR1,P#14.0];
MWJ0: NOP   0;
NETWORK
TITLE = Prepare Control Byte
      SET;
      R     #Snd.Control.Mbx;
      LAR1  P##Snd;
      L     DIW [AR1,P#0.0];
      LAR1  #tmpAddrIO;
      T     QW [AR1,P#0.0];
NETWORK
TITLE = Status/ StMode ASI Master
      A     #OutDPFault;
      =     #Fault.DPMaster;
      A     #Fault.ASIMaster;
      =     #Fault.ASIMaster;
      A     #Rcv.Status.Overflow;
      =     #Fault.Overflow;
      A     #Rcv.Status.ASIInactive;
      =     #Fault.ASIInactive;
      A     #Rcv.Status.ErrPower;
      =     #Fault.ErrPower;
      A     #Rcv.Status.ErrMapping;
      =     #Fault.ErrMapping;
      A     #Rcv.Status.ErrGeneral;
      =     #Fault.ErrGeneral;
//----------
      A     #Fault.DPMaster;
      O     #Fault.ASIMaster;
      O     #Fault.Overflow;
      O     #Fault.ASIInactive;
      O     #Fault.ErrPower;
      O     #Fault.ErrMapping;
      =     #tmpRelavantFaultSlaves;
      A     #tmpRelavantFaultSlaves;
      O     #Fault.ErrGeneral;
      =     #OutFaultRelevant;
//=======================================
//State
      AN    #OutFaultRelevant;
      =     #StOk;
      A     #OutFaultRelevant;
      =     #StFault;
//=======================================
//Test Log Message
      AN    #StFault;
      A     #OutMsgDone;
      JC    MSGO;
      A     #StFault;
      AN    #InLogOff;
      AN    #Par.ParLogOff;
      AN    #OutMsgDone;
      JC    MSCO;
      JU    MSST;	//-->StCode
//=======================================
//New Alarm
MSCO: S     #OutMsgDone;
      A     #InHornOff;
      JC    MSH2;
      CALL  "SYS_Horn_Code" (
           FcCode                   := 1,
           ParObjectType            := 1899,
           ParObjectNo              := #Par.ParObjectNo,
           ParHornCode              := #Par.ParHornCode);
MSH2: L     B#(1, 211);	//[1.1] ASI Master Alarm Coming 
      JU    MSLG;
//=======================================
//Alarm Going
MSGO: R     #OutMsgDone;
      L     B#(3, 212);	//[1.1] ASI Master Alarm Going 
//=======================================
//Entry Log Message
MSLG: T     #tmpLOGvalue;
      T     #OutAlarmNoLog;
      CALL  "GCS7_LogConvert" (
           ObjectNo                 := #Par.ParObjectNo,
           MsgType                  := #Par.ParMsgType,
           ClassMsgTxt              := #tmpLOGvalue,
           OType                    := 1899);	// LOG Message Converter / Entry / Contains Class and TextNo
//=======================================
//StCode
MSST: A     #StOk;
      L     2;	// StOk
      JC    MSSC;
      A     #Fault.DPMaster;
      L     33;	// StFault.DPMaster
      JC    MSSC;
      A     #Fault.ASIMaster;
      L     34;	// StFault.ASIMaster
      JC    MSSC;
      A     #Fault.Overflow;
      L     38;	// StFault.Overflow
      JC    MSSC;
      A     #Fault.ASIInactive;
      L     39;	// StFault.ASIInactive
      JC    MSSC;
      A     #Fault.ErrPower;
      L     40;	// StFault.ErrPower
      JC    MSSC;
      A     #Fault.ErrMapping;
      L     41;	// StFault.ErrMapping
      JC    MSSC;
      A     #Fault.ErrGeneral;
      L     42;	// StFault.ErrGeneral
      JC    MSSC;
      L     34;	// StFault.ASIMaster
MSSC: T     #StCode;
NETWORK
TITLE = Status/StCode Slave
      L     P##Slaves;
      T     #tmpAddr;
      L     1;
SLLP: T     #tmpIdx;
      L     63;
      >I;
      JC    SLJ0;
//=======================================
//Copy Data of SlavesA[x] to tmpSlave
      LAR1  #tmpAddr;
      L     DID [AR1,P#0.0];
      LAR1  P##tmpSlave;
      T     DID [AR1,P#0.0];
      LAR1  #tmpAddr;
      L     DID [AR1,P#4.0];
      LAR1  P##tmpSlave;
      T     DID [AR1,P#4.0];
//=======================================
//Copy Bit Information to tmpSlave 
      LAR1  P##Slaves_Detected;
      L     #tmpIdx;
      +AR1;
      A     DIX [AR1,P#0.0];	//Slaves_Detected
      =     #tmpSlave.OutDetected;
      A     DIX [AR1,P#8.0];	//Slaves_CfgDiff
      =     #tmpSlave.OutCfgDiff;
      A     DIX [AR1,P#16.0];	//Slaves_PeripheralFault
      =     #tmpSlave.OutPeripheralFault;
      A     DIX [AR1,P#24.0];	//Slaves_Corrupted
      =     #tmpSlave.OutCorrupted;
//=======================================
      A     #tmpSlave.Par.ParDIDO;
      O     #tmpSlave.Par.ParAI;
      O     #tmpSlave.Par.ParAO;
      =     #tmpUsed;
//=======================================
//Summary State
      A     #tmpSlave.OutDetected;
      AN    #tmpSlave.OutCfgDiff;
      AN    #tmpSlave.OutPeripheralFault;
      AN    #tmpSlave.OutCorrupted;
      AN    #tmpRelavantFaultSlaves;	//ASI Master
      A     #tmpUsed;
      =     #tmpSlave.StOk;
      AN    #tmpSlave.StOk;
      =     #tmpSlave.StFault;
      =     DIX [AR1,P#32.0];	//SlavesX_Faulted
//=======================================
//Test Log Message
      AN    #tmpUsed;
      JC    SLST;	//-->StCode
      AN    #tmpSlave.StFault;
      A     #tmpSlave.OutMsgDone;
      JC    SLGO;
      A     #tmpSlave.StFault;
      AN    #tmpRelavantFaultSlaves;
      AN    #InLogOff;
      AN    #Par.ParLogOff;
      AN    #tmpSlave.OutMsgDone;
      JC    SLCO;
      JU    SLST;	//-->StCode
//=======================================
//New Alarm
SLCO: S     #tmpSlave.OutMsgDone;
      A     #InHornOff;
      JC    SLH2;
      CALL  "SYS_Horn_Code" (
           FcCode                   := 1,
           ParObjectType            := 1899,
           ParObjectNo              := #Par.ParObjectNo,
           ParHornCode              := #Par.ParHornCode);
SLH2: L     B#(1, 0);	//ASI Slave Alarm Coming 
      JU    SLLG;
//=======================================
//Alarm Going
SLGO: R     #tmpSlave.OutMsgDone;
      L     B#(3, 0);	//ASI Slave Alarm Going
//=======================================
//Entry Log Message
SLLG: T     #tmpLOGvalue;
      L     31;
      L     #tmpIdx;
      >=I;
//[1.1]       SPB   SLLL
      JC    LOG1;	//[1.1] 
//Message Slave B
      L     100;
      L     #tmpIdx;
      +I;
      L     32;
      -D;
      JU    LOG1;
//Message Slave A
//[1.1] SLLL: L     100
//[1.1]       L     #tmpIdx
//[1.1]       +I    
//=======================================
//Entry Log Message
LOG1: A     #tmpSlave.OutMsgDone;	//[1.1]
      JC    LOG2;	//[1.1]
      L     40;	//[1.1]
      +I;	//[1.1]
LOG2: L     #tmpLOGvalue;	//[1.1]
      +I;
      T     #tmpLOGvalue;
      T     #OutAlarmNoLog;
      CALL  "GCS7_LogConvert" (
           ObjectNo                 := #Par.ParObjectNo,
           MsgType                  := #Par.ParMsgType,
           ClassMsgTxt              := #tmpLOGvalue,
           OType                    := 1899);	// LOG Message Converter / Entry / Contains Class and TextNo
//=======================================
//StCode
SLST: AN    #tmpUsed;
      L     0;	// StNotUsed
      JC    SLSC;
      A     #tmpSlave.StOk;
      L     2;	// StOk
      JC    SLSC;
      A     #Fault.DPMaster;
      L     33;	// StFault.DPMaster
      JC    SLSC;
      A     #tmpSlave.OutCfgDiff;
      L     35;	// StFault.CfgDiff
      JC    SLSC;
      A     #tmpSlave.OutPeripheralFault;
      L     36;	// StFault.PeripheralFault
      JC    SLSC;
      A     #tmpSlave.OutCorrupted;
      L     37;	// StFault.Corrupted
      JC    SLSC;
      A     #tmpRelavantFaultSlaves;
      L     34;	// StFault.ASIMaster
      JC    SLSC;
      L     32;	// StFault
SLSC: T     #tmpSlave.StCode;
//=======================================
//Copy Data oftmpSlave to  SlavesA[x] to 
      LAR1  P##tmpSlave;
      L     DID [AR1,P#0.0];
      LAR1  #tmpAddr;
      T     DID [AR1,P#0.0];
      LAR1  P##tmpSlave;
      L     DID [AR1,P#4.0];
      LAR1  #tmpAddr;
      T     DID [AR1,P#4.0];
//=======================================
//Pointer to Next Slave
      L     #tmpAddr;
      L     #tmpLenSlaveData;
      +D;
      T     #tmpAddr;
      L     #tmpIdx;
      +     1;
      JU    SLLP;
//=======================================
SLJ0: NOP   0;
NETWORK
TITLE = Copy Slaves_Faulted to  "SSA_SYS_ASI_Info"
      L     1;
      L     #Par.ParASIMasterIdx;
      >I;
      BEC;
      +     -1;
      L     P#8.0;
      *D;
      T     #tmpAddr;	//Address  "SSA_SYS_ASI_Info".Master[x]
      OPN   "SSA_SYS_ASI_Info";
      LAR1  P##Slaves_Faulted;
      L     DID [AR1,P#0.0];	//  Slaves_Faulted.A
      LAR1  #tmpAddr;
      T     DBD [AR1,P#0.0];	//  "SSA_SYS_ASI_Info".Master[x].Slaves_Faulted.A
      LAR1  P##Slaves_Faulted;
      L     DID [AR1,P#4.0];	//  Slaves_Faulted.B
      LAR1  #tmpAddr;
      T     DBD [AR1,P#4.0];	//  "SSA_SYS_ASI_Info".Master[x].Slaves_Faulted.B
END_FUNCTION_BLOCK

FUNCTION_BLOCK "COM_PLCSend"	// FB 1701
//COPYRIGHT:    (C) 1997 BY  BUHLER LTD.
//                           CH-9240 UZWIL  SWITZERLAND
//
//PRODUCT:      Project
//
//TITLE:        Send Data PLC --> PLC
//
//-------------------------------------------------------------------------
//
//IDENT:        AUTHOR:             DEPT:                       DATE:
//
//FB1701.1.2     A.Egli              CT3                        24-Nov-2004
//              Monitoring timeout send
//FB701.1.1     A.Egli              CT3                         4-Mar-2002
//              Slow down communication
//FB701.1A      A.Egli              AEE61                       7-Jul-1997
//              1st Release in S7
//
//-------------------------------------------------------------------------
//
//PURPOSE:      In a loop this modul send data blocks form one PLC
//              to a remote PLC.
//              On the remote PLC you must call the FB702 to read the data.
//
//RESTRICTIONS: S7
//
//-------------------------------------------------------------------------
//
//
//ID        : Communication ID            
//
//
AUTHOR : EA
FAMILY : PLCCom
NAME : SendPLC
VERSION : 1.2
VAR_INPUT
  ID : WORD ;	//Communication ID
  DB_SendData : INT ;	//DB Number
  DBB_SendData : INT ;	//1st byte
  Len_SendData : INT ;	//Lenght in byte
  ParMaxTimeOutSnd : INT ;	//[s]
  ParAutoSendIntervall : INT ;	//[s]
  ParMaxCycleTime : INT ;	//[ms]
  ParNoTimeOut : INT ;	//[number]]
END_VAR
VAR_IN_OUT
  SndOwnCounter : DINT ;
  SndPartnerCounterCopy : DINT ;
  RcvPartnerCounter : DINT ;
  RcvOwnCounterCopy : DINT ;
END_VAR
VAR
  CmdSend : BOOL ;
  InComSimulation : BOOL ;
  spare2 : BOOL ;
  spare3 : BOOL ;
  spare4 : BOOL ;
  spare5 : BOOL ;
  spare6 : BOOL ;
  CmdErrorSaved : BOOL ;
  CmdDone : BOOL ;
  CmdError : BOOL ;
  OutCfgFault : BOOL ;
  CmdCopied : BOOL ;
  OutChange : BOOL ;	//Send data has changed
  OutComRunning : BOOL ;
  PulseComPlcRunning : BOOL ;
  OutTimeOut : INT ;
  OutSendIntervall : INT ;
  Watchdog : STRUCT
   infCycleTimeOk : BOOL ;
   outCommRunning : BOOL ;
   EdgeComPlcRunning : BOOL ;
   intActCycleTime : INT ;
   intActNoTimeOut : INT ;
   intDelayTimeComOK : INT ;
  END_STRUCT ;
  BSND : SFB 12;
  SndDataBuffer : ARRAY  [1 .. 512 ] OF INT ;
END_VAR
VAR_TEMP
  tmpDB : INT ;
  tmpByte : INT ;
  tmpLen : INT ;
  tmpAddrRead : DWORD ;
  tmpAddrWrite : DWORD ;
  tmpCompare : BOOL ;
  tmpLenConvert : WORD ;
  tmpFlagSend : BOOL ;
  tmpCnt : INT ;
  tmpCycleTimeOk : BOOL ;
END_VAR
BEGIN
NETWORK
TITLE = WD Watchdog: Copy counter
//Receiverd Counter must be copied to send data
      L     #RcvPartnerCounter;
      T     #SndPartnerCounterCopy;
NETWORK
TITLE = WD Watchdog (1)
      AN    "SYS_Scan0_Tick100ms";
      JC    WD00;
// 
//-Calculate cycle time [ms]---
      L     #SndOwnCounter;
      L     #RcvOwnCounterCopy;
      -D;
      L     L#100;
      *D;
      T     #Watchdog.intActCycleTime;
      L     #ParMaxCycleTime;
      <=D;
      =     #tmpCycleTimeOk;
// 
//-Increment counter---
      L     #SndOwnCounter;
      +     L#1;
      T     #SndOwnCounter;
      L     0;
      <D;
      JCN   WD01;
      L     0;
      T     #SndOwnCounter;
      JU    WD01;
// 
//-Check cycle time---
WD01: A     #tmpCycleTimeOk;
      JCN   WD02;
      L     0;
      T     #Watchdog.intActNoTimeOut;
      JU    WD03;
// 
//-Increment time out counter---
WD02: A     #Watchdog.infCycleTimeOk;
      JCN   WD03;
      L     #Watchdog.intActNoTimeOut;
      +     1;
      T     #Watchdog.intActNoTimeOut;
// 
//-Check if number of retrys are exeeded---
WD03: L     #ParNoTimeOut;
      L     #Watchdog.intActNoTimeOut;
      >=I;
      =     #Watchdog.infCycleTimeOk;
// 
//-Delay reset of intCycleTimeOut---
      A     #Watchdog.infCycleTimeOk;
      JC    WD04;
      R     #Watchdog.outCommRunning;
      L     0;
      T     #Watchdog.intDelayTimeComOK;
      JU    WD05;
WD04: L     2000;	//[ms]
      L     #Watchdog.intDelayTimeComOK;
      <=I;
      S     #Watchdog.outCommRunning;
      JC    WD05;
      AN    "SYS_Scan0_Tick100ms";
      JC    WD05;
      +     100;	//100ms
      T     #Watchdog.intDelayTimeComOK;
//-----------------------------------  
//OutCommRunning 
WD05: A     #Watchdog.outCommRunning;
      O     #InComSimulation;
      =     #OutComRunning;
//-Edges---
      A     #OutComRunning;
      FP    #Watchdog.EdgeComPlcRunning;
      =     #PulseComPlcRunning;
WD00: NOP   0;
NETWORK
TITLE = Simulation
      A     #InComSimulation;
      BEC;
NETWORK
TITLE = ParMaxTimeOutSnd [1.2]
//[1.2] This function is moved to this netzwerk
      AN    "SYS_Tick1s";	//[1.2]
      ON    #BSND.REQ;	//[1.2]
      JC    MOJ0;	//[1.2]
      L     #OutTimeOut;	//[1.2]
      +     1;	//[1.2]
      T     #OutTimeOut;	//[1.2]
      L     #ParMaxTimeOutSnd;	//[1.2]
      <I;	//[1.2]
      JC    MOJ0;	//[1.2]
      R     #BSND.REQ;	//[1.2]
      S     #CmdSend;	//[1.2]
MOJ0: NOP   0;	//[1.2] 
NETWORK
TITLE = SendIntevall
      AN    "SYS_Tick1s";
      JC    X1;
      L     #OutSendIntervall;
      +     1;
      T     #OutSendIntervall;
      L     #ParAutoSendIntervall;
      >=I;
      S     #CmdSend;
X1:   NOP   0;
      AN    "GCS7_Gr_OutTick500ms";
      BEC;
NETWORK
TITLE = Test Telegramm Done
//Set address send buffer
      CLR;
      =     #tmpFlagSend;
Send: L     #Len_SendData;
      T     #tmpLenConvert;
      L     #ID;
      T     #BSND.ID;
      BLD   16;
      =     L 29.0;
      L     DINO;
      T     LW 27;
      CDB;
      OPN   DI [LW 27];
      TAR2  LD 23;
      L     W#16#1002;
      T     DIW [AR2,P#58.0];
      L     1024;
// Check answer
      T     DIW [AR2,P#60.0];
      L     DBNO;
      T     DIW [AR2,P#62.0];
      +AR2  P#72.0;
      TAR2;
      LAR2  LD 23;
      T     DID [AR2,P#64.0];
      L     #tmpLenConvert;
      T     #BSND.LEN;
      +AR2  P#46.0;	// [1.1]
      UC    "SIEMENS_BSEND";
      LAR2  LD 23;
      L     #BSND.LEN;
      T     #tmpLenConvert;	// [1.2]
      CDB;	// [1.2]
      BLD   17;
      A     #BSND.DONE;
      S     #CmdDone;
      R     #CmdError;
      R     #BSND.REQ;
      BEC;
      A     #BSND.ERROR;
      R     #BSND.ERROR;
      R     #BSND.REQ;
      S     #CmdError;
      S     #CmdErrorSaved;
      R     #CmdDone;
      S     #CmdCopied;
      BEC;
      A     #BSND.REQ;
      BEC;
NETWORK
TITLE = Prepare Send Telegram
      A     #CmdCopied;
      R     #CmdCopied;
//[1.1]      S     #BSND.REQ; 
      JC    Do;
      A     #CmdSend;
      R     #CmdSend;
      JC    Copy;
      L     #DB_SendData;
      T     #tmpDB;
      OPN   DB [#tmpDB];
      L     #DBB_SendData;
      SLD   3;
      T     #tmpAddrRead;
      L     P##SndDataBuffer;
      T     #tmpAddrWrite;
      L     #Len_SendData;
      T     #tmpCnt;
LOOP: L     DBW [#tmpAddrRead];
      L     DIW [#tmpAddrWrite];
      <>I;
      JC    Copy;
      L     #tmpAddrRead;
      +     L#16;
      T     #tmpAddrRead;
      L     #tmpAddrWrite;
      +     L#16;
      T     #tmpAddrWrite;
      L     #tmpCnt;
      +     -2;
      T     #tmpCnt;
      L     0;
      >I;
      JC    LOOP;
      BEC;
//Copy Send Data 
Copy: L     DINO;
      T     #tmpDB;
      L     P##SndDataBuffer;
      L     DW#16#FFFFF;
      AD;
      SRD   3;
      T     #tmpByte;
      CALL  "SYS_Copy_DBtoDB" (
           DBSource                 := #DB_SendData,
           ByteSource               := #DBB_SendData,
           DBDest                   := #tmpDB,
           ByteDest                 := #tmpByte,
           NoOfByte                 := #Len_SendData,
           Fault                    := #OutCfgFault);
      SET;
      S     #CmdCopied;
Do:   L     0;
      T     #OutTimeOut;
      T     #OutSendIntervall;
      SET;
      A     "GCS7_Gr_OutTick500ms";	//[1.1]
      S     #BSND.REQ;	//[1.1]
      AN    #tmpFlagSend;
      S     #tmpFlagSend;
      JC    Send;
NETWORK
TITLE = Save
      NOP   0;
END_FUNCTION_BLOCK

FUNCTION_BLOCK "COM_PLCReceive"	// FB 1702
//COPYRIGHT:    (C) 1997 BY  BUHLER LTD.
//                           CH-9240 UZWIL  SWITZERLAND
//
//PRODUCT:      Project
//
//TITLE:        Send Data PLC --> PLC
//
//-------------------------------------------------------------------------
//
//IDENT:        AUTHOR:             DEPT:                       DATE:
//
//FB7.1A        A.Egli              AEE61                       7-Jul-1997
//              1st Release in S7
//
//-------------------------------------------------------------------------
//
//PURPOSE:      In a loop this modul send data blocks form one PLC
//              to a remote PLC.
//              On the remote PLC you must call the FB702 to read the data.
//
//RESTRICTIONS: S7
//
//-------------------------------------------------------------------------
//
//
//ID        : Communication ID            
//
//
AUTHOR : EA
FAMILY : PLCCom
NAME : SendPLC
VERSION : 0.1
VAR_INPUT
  ID : WORD ;	//Communication ID
  DB_RcvData : INT ;
  DBB_RcvData : INT ;
  Len_RcvData : INT ;
  MaxTimeOutRcv : INT  := 10;	//[s]
END_VAR
VAR
  spare0 : BOOL ;
  spare1 : BOOL ;
  spare2 : BOOL ;
  spare3 : BOOL ;
  spare4 : BOOL ;
  spare5 : BOOL ;
  spare6 : BOOL ;
  spare7 : BOOL ;
  CmdDone : BOOL ;
  CmdError : BOOL ;
  OutCfgFault : BOOL ;
  spare13 : BOOL ;
  OutTimeOutRcv : BOOL ;
  OutTimeOutAc : INT ;
  BRCV : SFB 13;
  RcvDataBuffer : ARRAY  [1 .. 512 ] OF INT ;
END_VAR
VAR_TEMP
  tmpDB : INT ;
  tmpByte : INT ;
  tmpLen : INT ;
  tmpAddrRead : DWORD ;
  tmpAddrWrite : DWORD ;
  tmpCompare : BOOL ;
  tmpLenConvert : WORD ;
  tmpFlagSend : BOOL ;
  tmpCnt : INT ;
END_VAR
BEGIN
NETWORK
TITLE = Convert
NETWORK
TITLE = Test Telegramm Done
      CLR;
      =     #tmpFlagSend;
      SET;
      S     #BRCV.EN_R;
      L     #ID;
      T     #BRCV.ID;
      BLD   16;
      =     L 28.0;
      L     DINO;
      T     LW 26;
      CDB;
      OPN   DI [LW 26];
      TAR2  LD 22;
      L     W#16#1002;
      T     DIW [AR2,P#26.0];
// Check answer
      L     1024;
      T     DIW [AR2,P#28.0];
      L     DBNO;
      T     DIW [AR2,P#30.0];
      +AR2  P#40.0;
      TAR2;
      LAR2  LD 22;
      T     DID [AR2,P#32.0];
      +AR2  P#14.0;
      UC    "SIEMENS_BRCV";
      LAR2  LD 22;
      CDB;
      BLD   17;
      A     #BRCV.NDR;
      R     #BRCV.NDR;
      S     #CmdDone;
      R     #CmdError;
      JC    Copy;
      A     #BRCV.ERROR;
      R     #BRCV.ERROR;
      S     #CmdError;
      R     #CmdDone;
      BEC;
      AN    "SYS_Tick1s";
      BEC;
      L     #OutTimeOutAc;
      +     1;
      T     #OutTimeOutAc;
      L     #MaxTimeOutRcv;
      <I;
      BEC;
      S     #OutTimeOutRcv;
      BEU;
NETWORK
TITLE = Read data
Copy: R     #OutTimeOutRcv;
      L     0;
      T     #OutTimeOutAc;
      L     DINO;
      T     #tmpDB;
      L     P##RcvDataBuffer;
      L     DW#16#FFFFF;
      AD;
      SRD   3;
      T     #tmpByte;
      CALL  "SYS_Copy_DBtoDB" (
           DBSource                 := #tmpDB,
           ByteSource               := #tmpByte,
           DBDest                   := #DB_RcvData,
           ByteDest                 := #DBB_RcvData,
           NoOfByte                 := #Len_RcvData,
           Fault                    := #OutCfgFault);
END_FUNCTION_BLOCK

